KUKA KRL program: MyProgram_320().src

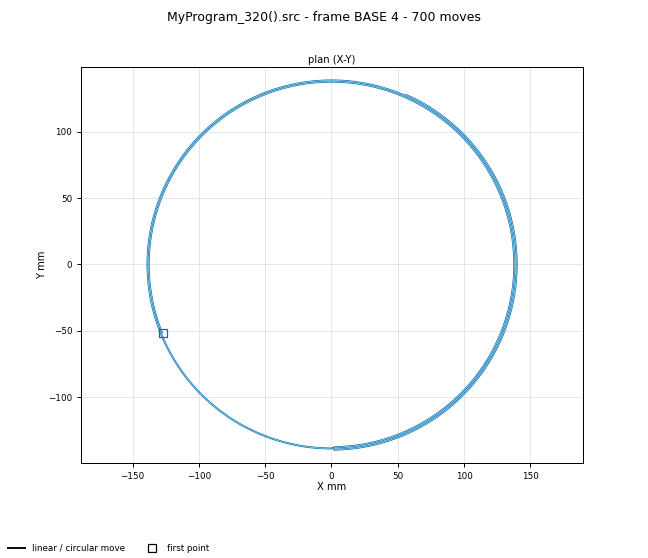
[picture p0: tool path of MyProgram_320().src in frame BASE 4, 700 of 700 moves have a stored position in this frame; points joined in program order, loops and branches not executed]
&ACCESS RVP
&REL 1
&PARAM TEMPLATE = C:\KRC\Roboter\Template\vorgabe
&PARAM EDITMASK = *
DEF MyProgram_320()
; ---- Setting reference (Base) ----
$BASE = BASE_DATA[4]

; --------------------------
; ---- Setting tool (TCP) ----
$TOOL = TOOL_DATA[3]
; --------------------------

$VEL.CP = VEL_APROX_PRINT
Startdeposition()
$VEL.CP = VEL_PRINT
LIN {X -127.2206,Y -51.8172,Z 185,A -153.9246,B 3.1278,C 0.2354,E1 2.9885,E2 247.0767} C_DIS
LIN {X -128.3074,Y -49.0677,Z 185,A -155.3949,B 3.128,C 0.2331,E1 2.987,E2 248.577} C_DIS
LIN {X -129.8881,Y -44.7108,Z 185,A -157.1036,B 3.1284,C 0.2271,E1 2.9854,E2 250.256} C_DIS
LIN {X -131.3839,Y -40.1019,Z 185,A -159.2672,B 3.1288,C 0.2223,E1 2.9836,E2 252.4369} C_DIS
LIN {X -132.2695,Y -37.0766,Z 185,A -160.5831,B 3.129,C 0.2188,E1 2.9825,E2 253.7523} C_DIS
LIN {X -133.0577,Y -34.142,Z 185,A -162.0522,B 3.1292,C 0.2162,E1 2.9815,E2 255.2465} C_DIS
LIN {X -133.9039,Y -30.6537,Z 185,A -163.578,B 3.1295,C 0.2122,E1 2.9805,E2 256.7752} C_DIS
LIN {X -134.6157,Y -27.3594,Z 185,A -164.9526,B 3.1298,C 0.2082,E1 2.9797,E2 258.145} C_DIS
LIN {X -135.1791,Y -24.4249,Z 185,A -166.2419,B 3.13,C 0.205,E1 2.979,E2 259.4392} C_DIS
LIN {X -135.7212,Y -21.207,Z 185,A -167.7582,B 3.1302,C 0.2018,E1 2.9784,E2 260.9744} C_DIS
LIN {X -136.2012,Y -17.8658,Z 185,A -169.3042,B 3.1304,C 0.1984,E1 2.9778,E2 262.5371} C_DIS
LIN {X -136.7019,Y -13.5167,Z 185,A -171.2437,B 3.1307,C 0.1937,E1 2.9772,E2 264.4899} C_DIS
LIN {X -136.999,Y -10.063,Z 185,A -172.73,B 3.1309,C 0.1898,E1 2.9768,E2 265.9804} C_DIS
LIN {X -137.2502,Y -5.6994,Z 185,A -174.6658,B 3.1312,C 0.1851,E1 2.9766,E2 267.9293} C_DIS
LIN {X -137.3622,Y -1.4594,Z 185,A -176.5532,B 3.1315,C 0.1806,E1 2.9765,E2 269.8305} C_DIS
LIN {X -137.346,Y 2.474,Z 185,A -178.1887,B 3.1317,C 0.1759,E1 2.9765,E2 271.4643} C_DIS
LIN {X -137.2122,Y 6.5512,Z 185,A 179.9992,B 3.132,C 0.1716,E1 2.9767,E2 273.2891} C_DIS
LIN {X -136.9944,Y 10.1259,Z 185,A 178.4827,B 3.1322,C 0.1674,E1 2.977,E2 274.8074} C_DIS
LIN {X -136.6818,Y 13.7268,Z 185,A 176.7446,B 3.1324,C 0.1641,E1 2.9775,E2 276.5735} C_DIS
LIN {X -136.1552,Y 18.2164,Z 185,A 174.8363,B 3.1326,C 0.1589,E1 2.9781,E2 278.4833} C_DIS
LIN {X -135.5392,Y 22.3415,Z 185,A 173.1558,B 3.1329,C 0.1538,E1 2.9789,E2 280.1551} C_DIS
LIN {X -134.953,Y 25.6446,Z 185,A 171.7399,B 3.1331,C 0.15,E1 2.9796,E2 281.5721} C_DIS
LIN {X -134.4845,Y 28.0041,Z 185,A 170.5079,B 3.1331,C 0.1481,E1 2.9803,E2 282.832} C_DIS
LIN {X -133.7699,Y 31.2406,Z 185,A 169.0156,B 3.1333,C 0.1447,E1 2.9812,E2 284.3369} C_DIS
LIN {X -132.7902,Y 35.167,Z 185,A 167.5567,B 3.1336,C 0.1392,E1 2.9822,E2 285.766} C_DIS
LIN {X -131.8831,Y 38.4286,Z 185,A 165.6724,B 3.1336,C 0.1372,E1 2.9837,E2 287.708} C_DIS
LIN {X -130.4216,Y 43.1295,Z 185,A 163.8308,B 3.1339,C 0.1309,E1 2.9852,E2 289.5218} C_DIS
LIN {X -129.6058,Y 45.525,Z 185,A 162.5514,B 3.134,C 0.1289,E1 2.9864,E2 290.8282} C_DIS
LIN {X -128.1871,Y 49.3771,Z 185,A 161.0189,B 3.1342,C 0.1238,E1 2.9879,E2 292.3371} C_DIS
LIN {X -127.3534,Y 51.4877,Z 185,A 158.726,B 3.1342,C 0.1265,E1 2.9906,E2 294.7944} C_DIS
LIN {X -124.3017,Y 58.4774,Z 185,A 156.4051,B 3.1346,C 0.1151,E1 2.9931,E2 297.0081} C_DIS
LIN {X -122.5678,Y 62.0248,Z 185,A 154.87,B 3.1347,C 0.1105,E1 2.995,E2 298.5281} C_DIS
LIN {X -120.8252,Y 65.3591,Z 185,A 153.0785,B 3.1348,C 0.1075,E1 2.9974,E2 300.3459} C_DIS
LIN {X -118.619,Y 69.2824,Z 185,A 151.1069,B 3.135,C 0.1033,E1 3.0001,E2 302.3275} C_DIS
LIN {X -116.2679,Y 73.1587,Z 185,A 149.325,B 3.1351,C 0.0984,E1 3.0027,E2 304.0945} C_DIS
LIN {X -113.2304,Y 77.7771,Z 185,A 146.7901,B 3.1353,C 0.094,E1 3.0067,E2 306.6559} C_DIS
LIN {X -110.5879,Y 81.4907,Z 185,A 144.8026,B 3.1353,C 0.0901,E1 3.0099,E2 308.6525} C_DIS
LIN {X -107.9657,Y 84.9341,Z 185,A 142.9194,B 3.1355,C 0.0865,E1 3.0132,E2 310.5437} C_DIS
LIN {X -104.5605,Y 89.0927,Z 185,A 140.5857,B 3.1355,C 0.0821,E1 3.0173,E2 312.8869} C_DIS
LIN {X -101.4653,Y 92.6032,Z 185,A 138.5535,B 3.1357,C 0.0785,E1 3.0212,E2 314.9274} C_DIS
LIN {X -98.4395,Y 95.8133,Z 185,A 136.6894,B 3.1357,C 0.0749,E1 3.0248,E2 316.793} C_DIS
LIN {X -95.2668,Y 98.9686,Z 185,A 134.7267,B 3.1358,C 0.0718,E1 3.0287,E2 318.766} C_DIS
LIN {X -92.1092,Y 101.9135,Z 185,A 132.8935,B 3.1359,C 0.0686,E1 3.0325,E2 320.6017} C_DIS
LIN {X -88.6534,Y 104.9339,Z 185,A 130.9144,B 3.1359,C 0.0655,E1 3.0367,E2 322.5872} C_DIS
LIN {X -86.0163,Y 107.1059,Z 185,A 129.2483,B 3.136,C 0.0643,E1 3.0404,E2 324.2815} C_DIS
LIN {X -83.4152,Y 109.1434,Z 185,A 128.0792,B 3.136,C 0.061,E1 3.0429,E2 325.4243} C_DIS
LIN {X -79.93,Y 111.721,Z 185,A 126.1941,B 3.1361,C 0.0585,E1 3.0472,E2 327.3174} C_DIS
LIN {X -76.2262,Y 114.2802,Z 185,A 124.3048,B 3.1361,C 0.0557,E1 3.0515,E2 329.2068} C_DIS
LIN {X -72.531,Y 116.6604,Z 185,A 122.6104,B 3.1362,C 0.0524,E1 3.0555,E2 330.8831} C_DIS
LIN {X -68.5121,Y 119.0656,Z 185,A 120.4438,B 3.1362,C 0.0509,E1 3.0608,E2 333.0742} C_DIS
LIN {X -64.7458,Y 121.1547,Z 185,A 117.9732,B 3.1362,C 0.0521,E1 3.0671,E2 335.6243} C_DIS
LIN {X -60.0472,Y 123.5509,Z 185,A 116.2413,B 3.1363,C 0.0471,E1 3.0712,E2 337.2988} C_DIS
LIN {X -56.4708,Y 125.2241,Z 185,A 114.8247,B 3.1363,C 0.0441,E1 3.0748,E2 338.6867} C_DIS
LIN {X -53.2256,Y 126.6372,Z 185,A 112.9364,B 3.1363,C 0.0449,E1 3.0798,E2 340.6235} C_DIS
LIN {X -50.1738,Y 127.8774,Z 185,A 111.996,B 3.1363,C 0.0412,E1 3.0821,E2 341.5109} C_DIS
LIN {X -47.5465,Y 128.8785,Z 185,A 110.5514,B 3.1363,C 0.0417,E1 3.0859,E2 342.9876} C_DIS
LIN {X -43.669,Y 130.242,Z 185,A 108.8857,B 3.1364,C 0.04,E1 3.0903,E2 344.6463} C_DIS
LIN {X -40.3704,Y 131.3017,Z 185,A 107.4297,B 3.1364,C 0.039,E1 3.0942,E2 346.1028} C_DIS
LIN {X -36.1258,Y 132.5345,Z 185,A 105.463,B 3.1364,C 0.0385,E1 3.0995,E2 348.0833} C_DIS
LIN {X -32.4216,Y 133.4871,Z 185,A 104.0145,B 3.1364,C 0.0367,E1 3.1034,E2 349.5132} C_DIS
LIN {X -29.6457,Y 134.1324,Z 185,A 102.663,B 3.1364,C 0.0371,E1 3.1071,E2 350.8836} C_DIS
LIN {X -25.59,Y 134.9634,Z 185,A 100.9801,B 3.1364,C 0.0361,E1 3.1117,E2 352.5604} C_DIS
LIN {X -21.1664,Y 135.7275,Z 185,A 99.211,B 3.1364,C 0.0348,E1 3.1166,E2 354.316} C_DIS
LIN {X -17.9099,Y 136.1954,Z 185,A 97.7627,B 3.1364,C 0.0349,E1 3.1206,E2 355.7728} C_DIS
LIN {X -12.6318,Y 136.7867,Z 185,A 94.5314,B 3.1364,C 0.0411,E1 3.13,E2 359.1239} C_DIS
LIN {X -5.4981,Y 137.2581,Z 185,A 92.5658,B 3.1364,C 0.0344,E1 3.1351,E2 360.9673} C_DIS
LIN {X 1.8136,Y 137.357,Z 185,A 89.5018,B 3.1364,C 0.0348,E1 3.1437,E2 364.0318} C_DIS
LIN {X 9.2316,Y 137.0596,Z 185,A 86.3024,B 3.1364,C 0.0363,E1 3.1526,E2 367.2424} C_DIS
LIN {X 15.1597,Y 136.5297,Z 185,A 83.5212,B 3.1364,C 0.0394,E1 3.1605,E2 370.0585} C_DIS
LIN {X 19.2177,Y 136.0172,Z 185,A 82.2725,B 3.1364,C 0.037,E1 3.1638,E2 371.2518} C_DIS
LIN {X 22.3777,Y 135.5331,Z 185,A 80.9467,B 3.1364,C 0.0376,E1 3.1674,E2 372.5762} C_DIS
LIN {X 25.7451,Y 134.9337,Z 185,A 79.5762,B 3.1364,C 0.0381,E1 3.1712,E2 373.9396} C_DIS
LIN {X 28.5414,Y 134.3708,Z 185,A 78.4896,B 3.1364,C 0.0381,E1 3.1741,E2 375.0134} C_DIS
LIN {X 31.7927,Y 133.6387,Z 185,A 76.9984,B 3.1364,C 0.04,E1 3.1782,E2 376.5164} C_DIS
LIN {X 35.2086,Y 132.7791,Z 185,A 75.5841,B 3.1364,C 0.0407,E1 3.182,E2 377.9236} C_DIS
LIN {X 38.3332,Y 131.9111,Z 185,A 74.2324,B 3.1364,C 0.0419,E1 3.1856,E2 379.275} C_DIS
LIN {X 41.6265,Y 130.9089,Z 185,A 72.8018,B 3.1364,C 0.0432,E1 3.1895,E2 380.7046} C_DIS
LIN {X 44.8549,Y 129.8381,Z 185,A 71.3415,B 3.1364,C 0.045,E1 3.1933,E2 382.1696} C_DIS
LIN {X 49.4529,Y 128.1577,Z 185,A 69.3854,B 3.1364,C 0.0465,E1 3.1984,E2 384.115} C_DIS
LIN {X 52.5735,Y 126.9096,Z 185,A 68.0035,B 3.1363,C 0.048,E1 3.202,E2 385.4942} C_DIS
LIN {X 55.8092,Y 125.52,Z 185,A 66.7765,B 3.1363,C 0.0479,E1 3.2051,E2 386.6917} C_DIS
LIN {X 58.9894,Y 124.0571,Z 185,A 65.1798,B 3.1363,C 0.0508,E1 3.2092,E2 388.3049} C_DIS
LIN {X 62.1187,Y 122.52,Z 185,A 63.7792,B 3.1363,C 0.0524,E1 3.2127,E2 389.6988} C_DIS
LIN {X 65.4146,Y 120.7953,Z 185,A 62.0738,B 3.1362,C 0.0558,E1 3.2169,E2 391.4229} C_DIS
LIN {X 69.3364,Y 118.5873,Z 185,A 60.2725,B 3.1362,C 0.058,E1 3.2213,E2 393.2149} C_DIS
LIN {X 73.2071,Y 116.2374,Z 185,A 58.4362,B 3.1361,C 0.0605,E1 3.2256,E2 395.0447} C_DIS
LIN {X 76.9789,Y 113.7746,Z 185,A 56.6058,B 3.1361,C 0.0632,E1 3.2299,E2 396.8692} C_DIS
LIN {X 80.6259,Y 111.2199,Z 185,A 54.8233,B 3.136,C 0.0657,E1 3.2339,E2 398.6426} C_DIS
LIN {X 84.0737,Y 108.6371,Z 185,A 53.0719,B 3.136,C 0.0685,E1 3.2378,E2 400.3886} C_DIS
LIN {X 87.511,Y 105.8878,Z 185,A 51.2684,B 3.1358,C 0.0716,E1 3.2417,E2 402.1882} C_DIS
LIN {X 91.1,Y 102.8163,Z 185,A 49.6038,B 3.1358,C 0.0727,E1 3.2451,E2 403.8156} C_DIS
LIN {X 93.7824,Y 100.3758,Z 185,A 47.9612,B 3.1358,C 0.0768,E1 3.2485,E2 405.4743} C_DIS
LIN {X 96.8021,Y 97.4666,Z 185,A 46.2566,B 3.1356,C 0.0799,E1 3.2519,E2 407.1737} C_DIS
LIN {X 99.6214,Y 94.5841,Z 185,A 44.7019,B 3.1356,C 0.0823,E1 3.2549,E2 408.7131} C_DIS
LIN {X 102.2276,Y 91.7602,Z 185,A 43.0242,B 3.1355,C 0.0864,E1 3.2581,E2 410.4003} C_DIS
LIN {X 105.1144,Y 88.4387,Z 185,A 41.2518,B 3.1354,C 0.0898,E1 3.2613,E2 412.1653} C_DIS
LIN {X 107.8952,Y 85.0239,Z 185,A 39.4783,B 3.1353,C 0.0934,E1 3.2644,E2 413.9314} C_DIS
LIN {X 110.6338,Y 81.4283,Z 185,A 37.6704,B 3.1352,C 0.097,E1 3.2674,E2 415.7303} C_DIS
LIN {X 113.1668,Y 77.8697,Z 185,A 35.9227,B 3.1351,C 0.1005,E1 3.2702,E2 417.4693} C_DIS
LIN {X 114.8292,Y 75.3968,Z 185,A 34.6044,B 3.1349,C 0.1042,E1 3.2722,E2 418.7973} C_DIS
LIN {X 116.6535,Y 72.5421,Z 185,A 32.6213,B 3.1346,C 0.113,E1 3.2753,E2 420.8509} C_DIS
LIN {X 119.8789,Y 67.0784,Z 185,A 30.7963,B 3.1346,C 0.1118,E1 3.2776,E2 422.5758} C_DIS
LIN {X 122.1471,Y 62.8512,Z 185,A 29.0018,B 3.1346,C 0.1148,E1 3.2799,E2 424.3453} C_DIS
LIN {X 123.6929,Y 59.7517,Z 185,A 27.4883,B 3.1344,C 0.1192,E1 3.2818,E2 425.8679} C_DIS
LIN {X 125.0111,Y 56.9438,Z 185,A 26.0373,B 3.1342,C 0.124,E1 3.2835,E2 427.3391} C_DIS
LIN {X 126.4267,Y 53.7295,Z 185,A 23.9921,B 3.1338,C 0.1335,E1 3.2858,E2 429.4566} C_DIS
LIN {X 129.0057,Y 47.1998,Z 185,A 22.0204,B 3.1338,C 0.1319,E1 3.2876,E2 431.311} C_DIS
LIN {X 130.2761,Y 43.5666,Z 185,A 20.5744,B 3.1338,C 0.1347,E1 3.2889,E2 432.7378} C_DIS
LIN {X 131.3256,Y 40.2925,Z 185,A 19.2721,B 3.1337,C 0.1372,E1 3.29,E2 434.0243} C_DIS
LIN {X 132.3115,Y 36.9264,Z 185,A 17.8228,B 3.1335,C 0.1411,E1 3.2911,E2 435.4725} C_DIS
LIN {X 133.1382,Y 33.8247,Z 185,A 16.5536,B 3.1334,C 0.144,E1 3.292,E2 436.7337} C_DIS
LIN {X 133.8617,Y 30.8387,Z 185,A 15.3424,B 3.1332,C 0.1469,E1 3.2928,E2 437.9367} C_DIS
LIN {X 134.4778,Y 28.0373,Z 185,A 14.0616,B 3.133,C 0.151,E1 3.2935,E2 439.2289} C_DIS
LIN {X 135.2029,Y 24.2921,Z 185,A 12.5685,B 3.1329,C 0.1544,E1 3.2943,E2 440.7104} C_DIS
LIN {X 135.9145,Y 19.9358,Z 185,A 11.0001,B 3.1327,C 0.1568,E1 3.2949,E2 442.2454} C_DIS
LIN {X 136.6326,Y 14.2037,Z 185,A 8.465,B 3.1323,C 0.1649,E1 3.2958,E2 444.7979} C_DIS
LIN {X 137.239,Y 5.9882,Z 185,A 5.1999,B 3.1319,C 0.1728,E1 3.2964,E2 448.0435} C_DIS
LIN {X 137.352,Y 2.1098,Z 185,A 3.8317,B 3.1318,C 0.1748,E1 3.2964,E2 449.3808} C_DIS
LIN {X 137.3445,Y -2.5652,Z 185,A 1.3682,B 3.1312,C 0.1855,E1 3.2964,E2 451.9109} C_DIS
LIN {X 137.1832,Y -7.1289,Z 185,A -0.0422,B 3.1312,C 0.1859,E1 3.2962,E2 453.2598} C_DIS
LIN {X 136.8906,Y -11.443,Z 185,A -1.7494,B 3.1309,C 0.19,E1 3.2958,E2 454.9559} C_DIS
LIN {X 136.4657,Y -15.7279,Z 185,A -3.9041,B 3.1304,C 0.1987,E1 3.2952,E2 457.1577} C_DIS
LIN {X 135.8556,Y -20.3391,Z 185,A -5.3709,B 3.1304,C 0.1993,E1 3.2946,E2 458.5656} C_DIS
LIN {X 135.2516,Y -24.02,Z 185,A -6.7383,B 3.1302,C 0.2018,E1 3.294,E2 459.9098} C_DIS
LIN {X 134.7097,Y -26.8975,Z 185,A -7.7917,B 3.1301,C 0.2035,E1 3.2934,E2 460.9425} C_DIS
LIN {X 133.992,Y -30.2682,Z 185,A -9.2727,B 3.1298,C 0.2079,E1 3.2925,E2 462.4302} C_DIS
LIN {X 133.1727,Y -33.6888,Z 185,A -10.7278,B 3.1295,C 0.2118,E1 3.2916,E2 463.8848} C_DIS
LIN {X 132.2958,Y -36.9825,Z 185,A -11.9845,B 3.1294,C 0.214,E1 3.2907,E2 465.1212} C_DIS
LIN {X 131.4704,Y -39.8192,Z 185,A -13.3051,B 3.1291,C 0.2183,E1 3.2896,E2 466.4543} C_DIS
LIN {X 130.5719,Y -42.6782,Z 185,A -14.4871,B 3.1289,C 0.221,E1 3.2886,E2 467.6285} C_DIS
LIN {X 129.3343,Y -46.2882,Z 185,A -15.9446,B 3.1287,C 0.2239,E1 3.2873,E2 469.0698} C_DIS
LIN {X 128.1113,Y -49.5722,Z 185,A -17.3701,B 3.1284,C 0.2274,E1 3.2859,E2 470.4918} C_DIS
LIN {X 126.7284,Y -53.0073,Z 185,A -18.8286,B 3.1282,C 0.2306,E1 3.2843,E2 471.9402} C_DIS
LIN {X 125.6739,Y -55.465,Z 185,A -19.9685,B 3.1279,C 0.2338,E1 3.283,E2 473.0843} C_DIS
LIN {X 124.0202,Y -59.0665,Z 185,A -21.4912,B 3.1277,C 0.2368,E1 3.2813,E2 474.5913} C_DIS
LIN {X 122.6016,Y -61.9584,Z 185,A -22.7609,B 3.1275,C 0.2395,E1 3.2797,E2 475.8526} C_DIS
LIN {X 120.8252,Y -65.3591,Z 185,A -24.7938,B 3.1269,C 0.2478,E1 3.2769,E2 477.943} C_DIS
LIN {X 118.6705,Y -69.1946,Z 185,A -26.2059,B 3.1269,C 0.2482,E1 3.275,E2 479.3017} C_DIS
LIN {X 116.4356,Y -72.8922,Z 185,A -27.8995,B 3.1266,C 0.2515,E1 3.2726,E2 480.9826} C_DIS
LIN {X 114.5094,Y -75.8825,Z 185,A -29.7412,B 3.126,C 0.2586,E1 3.2697,E2 482.8721} C_DIS
LIN {X 111.9579,Y -79.5988,Z 185,A -31.1758,B 3.126,C 0.2587,E1 3.2674,E2 484.2502} C_DIS
LIN {X 109.3387,Y -83.16,Z 185,A -32.9566,B 3.1257,C 0.2624,E1 3.2645,E2 486.0242} C_DIS
LIN {X 106.5413,Y -86.7146,Z 185,A -34.8528,B 3.1253,C 0.2668,E1 3.2612,E2 487.9233} C_DIS
LIN {X 103.8669,Y -89.9008,Z 185,A -36.8226,B 3.1248,C 0.2728,E1 3.2575,E2 489.9251} C_DIS
LIN {X 100.8615,Y -93.2604,Z 185,A -38.2429,B 3.1248,C 0.2725,E1 3.2549,E2 491.2868} C_DIS
LIN {X 97.7188,Y -96.5482,Z 185,A -40.1537,B 3.1245,C 0.2766,E1 3.2512,E2 493.201} C_DIS
LIN {X 94.2509,Y -99.9358,Z 185,A -42.0108,B 3.1242,C 0.2792,E1 3.2475,E2 495.038} C_DIS
LIN {X 90.5016,Y -103.3437,Z 185,A -44.0948,B 3.1239,C 0.2831,E1 3.2432,E2 497.1198} C_DIS
LIN {X 87.0714,Y -106.2497,Z 185,A -45.9866,B 3.1235,C 0.2868,E1 3.2391,E2 499.0153} C_DIS
LIN {X 83.0844,Y -109.3963,Z 185,A -47.8812,B 3.1234,C 0.2886,E1 3.235,E2 500.8821} C_DIS
LIN {X 79.2752,Y -112.1867,Z 185,A -49.8775,B 3.123,C 0.2924,E1 3.2304,E2 502.8834} C_DIS
LIN {X 75.5788,Y -114.7094,Z 185,A -51.6453,B 3.1228,C 0.2946,E1 3.2264,E2 504.6396} C_DIS
LIN {X 72.2271,Y -116.8495,Z 185,A -53.152,B 3.1227,C 0.2959,E1 3.2228,E2 506.1275} C_DIS
LIN {X 66.1107,Y -120.4156,Z 185,A -56.0363,B 3.1223,C 0.2999,E1 3.2159,E2 509.005} C_DIS
LIN {X 62.9846,Y -122.0792,Z 185,A -57.6575,B 3.122,C 0.3032,E1 3.2118,E2 510.6463} C_DIS
LIN {X 59.3361,Y -123.8914,Z 185,A -59.2521,B 3.1218,C 0.3046,E1 3.2078,E2 512.2282} C_DIS
LIN {X 55.6679,Y -125.5832,Z 185,A -60.9267,B 3.1216,C 0.3067,E1 3.2036,E2 513.9027} C_DIS
LIN {X 51.6723,Y -127.279,Z 185,A -62.5593,B 3.1216,C 0.3074,E1 3.1994,E2 515.5129} C_DIS
LIN {X 48.9659,Y -128.3467,Z 185,A -63.9601,B 3.1213,C 0.3104,E1 3.1957,E2 516.9395} C_DIS
LIN {X 45.2189,Y -129.7119,Z 185,A -65.5888,B 3.1211,C 0.312,E1 3.1914,E2 518.5646} C_DIS
LIN {X 40.8738,Y -131.1477,Z 185,A -67.3488,B 3.1211,C 0.3126,E1 3.1868,E2 520.3062} C_DIS
LIN {X 36.9918,Y -132.2932,Z 185,A -68.9133,B 3.1211,C 0.3132,E1 3.1826,E2 521.8553} C_DIS
LIN {X 33.931,Y -133.1113,Z 185,A -70.292,B 3.1208,C 0.3148,E1 3.1789,E2 523.2424} C_DIS
LIN {X 30.5431,Y -133.9292,Z 185,A -71.7431,B 3.1208,C 0.316,E1 3.1749,E2 524.6941} C_DIS
LIN {X 26.6507,Y -134.7599,Z 185,A -73.4339,B 3.1206,C 0.3174,E1 3.1703,E2 526.39} C_DIS
LIN {X 23.6785,Y -135.3127,Z 185,A -75.6824,B 3.1197,C 0.326,E1 3.1638,E2 528.7694} C_DIS
LIN {X 16.2323,Y -136.4055,Z 185,A -77.6627,B 3.1205,C 0.3187,E1 3.1587,E2 530.5987} C_DIS
LIN {X 9.1529,Y -137.0646,Z 185,A -80.9036,B 3.1201,C 0.322,E1 3.1495,E2 533.8778} C_DIS
LIN {X 2.2312,Y -137.35,Z 185,A -83.5784,B 3.1201,C 0.3211,E1 3.1421,E2 536.5256} C_DIS
LIN {X 2.2312,Y -137.35,Z 185,A -83.5784,B 3.1201,C 0.3211,E1 3.1421,E2 536.5256} C_DIS
Enddeposition()
LIN {X 0.9813,Y -138.2634,Z 185,A -83.5483,B 3.1297,C 0.3191,E1 3.1516,E2 536.4499} C_DIS
Startdeposition()
$VEL.CP = VEL_PRINT
LIN {X 4.1352,Y -138.2067,Z 185,A -82.1164,B 3.1298,C 0.3178,E1 3.1557,E2 535.0005} C_DIS
LIN {X 7.7208,Y -138.0547,Z 185,A -80.675,B 3.1298,C 0.3178,E1 3.1597,E2 533.5646} C_DIS
LIN {X 10.8511,Y -137.844,Z 185,A -79.3806,B 3.1299,C 0.3173,E1 3.1633,E2 532.2704} C_DIS
LIN {X 14.4758,Y -137.5087,Z 185,A -77.875,B 3.1299,C 0.3167,E1 3.1675,E2 530.7643} C_DIS
LIN {X 17.1717,Y -137.2,Z 185,A -76.7623,B 3.13,C 0.3162,E1 3.1706,E2 529.6526} C_DIS
LIN {X 20.8522,Y -136.687,Z 185,A -75.2123,B 3.1301,C 0.3152,E1 3.1748,E2 528.1002} C_DIS
LIN {X 25.6575,Y -135.867,Z 185,A -73.2312,B 3.1302,C 0.3142,E1 3.1803,E2 526.1233} C_DIS
LIN {X 28.873,Y -135.2201,Z 185,A -71.8856,B 3.1303,C 0.3133,E1 3.184,E2 524.7786} C_DIS
LIN {X 32.1482,Y -134.4789,Z 185,A -70.5233,B 3.1303,C 0.3125,E1 3.1877,E2 523.4194} C_DIS
LIN {X 35.3199,Y -133.681,Z 185,A -69.171,B 3.1305,C 0.3113,E1 3.1913,E2 522.0667} C_DIS
LIN {X 38.0462,Y -132.933,Z 185,A -67.8723,B 3.1307,C 0.3092,E1 3.1949,E2 520.7501} C_DIS
LIN {X 41.7685,Y -131.8085,Z 185,A -66.5596,B 3.1307,C 0.3101,E1 3.1983,E2 519.4767} C_DIS
LIN {X 44.4883,Y -130.9179,Z 185,A -65.2589,B 3.1308,C 0.3079,E1 3.2018,E2 518.1597} C_DIS
LIN {X 48.0865,Y -129.6374,Z 185,A -63.6729,B 3.131,C 0.3061,E1 3.2059,E2 516.5721} C_DIS
LIN {X 51.3902,Y -128.3633,Z 185,A -62.2604,B 3.1311,C 0.3049,E1 3.2096,E2 515.1661} C_DIS
LIN {X 54.6278,Y -127.0191,Z 185,A -60.8496,B 3.1313,C 0.3035,E1 3.2132,E2 513.7599} C_DIS
LIN {X 57.7327,Y -125.6384,Z 185,A -59.6462,B 3.1313,C 0.3035,E1 3.2162,E2 512.583} C_DIS
LIN {X 60.3884,Y -124.3863,Z 185,A -58.2622,B 3.1316,C 0.3003,E1 3.2198,E2 511.1758} C_DIS
LIN {X 63.5069,Y -122.8234,Z 185,A -56.7072,B 3.1319,C 0.2973,E1 3.2237,E2 509.6048} C_DIS
LIN {X 67.3646,Y -120.7507,Z 185,A -54.953,B 3.1321,C 0.2952,E1 3.228,E2 507.8575} C_DIS
LIN {X 71.1713,Y -118.5469,Z 185,A -53.1835,B 3.1323,C 0.2928,E1 3.2322,E2 506.0939} C_DIS
LIN {X 74.9206,Y -116.2137,Z 185,A -51.5093,B 3.1324,C 0.2912,E1 3.2361,E2 504.4393} C_DIS
LIN {X 78.1008,Y -114.1,Z 185,A -49.9155,B 3.1327,C 0.2885,E1 3.2398,E2 502.8427} C_DIS
LIN {X 81.5037,Y -111.6954,Z 185,A -48.2879,B 3.1329,C 0.2864,E1 3.2435,E2 501.2271} C_DIS
LIN {X 84.5715,Y -109.3902,Z 185,A -46.6821,B 3.1332,C 0.2833,E1 3.247,E2 499.618} C_DIS
LIN {X 87.8428,Y -106.7818,Z 185,A -45.0586,B 3.1334,C 0.2811,E1 3.2505,E2 498.0079} C_DIS
LIN {X 90.9521,Y -104.1452,Z 185,A -43.3668,B 3.1336,C 0.2778,E1 3.2541,E2 496.3144} C_DIS
LIN {X 94.1057,Y -101.3048,Z 185,A -41.7154,B 3.1339,C 0.2753,E1 3.2575,E2 494.676} C_DIS
LIN {X 96.9393,Y -98.5967,Z 185,A -40.1086,B 3.1341,C 0.2722,E1 3.2607,E2 493.0703} C_DIS
LIN {X 99.6517,Y -95.8553,Z 185,A -38.5217,B 3.1344,C 0.2689,E1 3.2638,E2 491.4836} C_DIS
LIN {X 102.6999,Y -92.5821,Z 185,A -36.7443,B 3.1347,C 0.2657,E1 3.2672,E2 489.7149} C_DIS
LIN {X 105.5902,Y -89.2713,Z 185,A -34.9767,B 3.135,C 0.2622,E1 3.2704,E2 487.953} C_DIS
LIN {X 108.0789,Y -86.2409,Z 185,A -33.3908,B 3.1353,C 0.2589,E1 3.2731,E2 486.371} C_DIS
LIN {X 110.8016,Y -82.7136,Z 185,A -31.7,B 3.1355,C 0.2562,E1 3.276,E2 484.6994} C_DIS
LIN {X 113.1584,Y -79.4592,Z 185,A -30.0798,B 3.1358,C 0.2527,E1 3.2786,E2 483.0839} C_DIS
LIN {X 115.5333,Y -75.9643,Z 185,A -28.3636,B 3.1361,C 0.2488,E1 3.2813,E2 481.3709} C_DIS
LIN {X 117.9476,Y -72.1589,Z 185,A -26.5817,B 3.1364,C 0.2451,E1 3.2839,E2 479.5988} C_DIS
LIN {X 120.0197,Y -68.6573,Z 185,A -24.9011,B 3.1367,C 0.241,E1 3.2862,E2 477.9177} C_DIS
LIN {X 122.0101,Y -65.0556,Z 185,A -23.3573,B 3.1369,C 0.2383,E1 3.2883,E2 476.3939} C_DIS
LIN {X 123.6155,Y -61.951,Z 185,A -21.9277,B 3.1372,C 0.2348,E1 3.2901,E2 474.9657} C_DIS
LIN {X 125.1925,Y -58.697,Z 185,A -20.5769,B 3.1373,C 0.2324,E1 3.2917,E2 473.6332} C_DIS
LIN {X 126.5706,Y -55.665,Z 185,A -19.2064,B 3.1376,C 0.2289,E1 3.2932,E2 472.2629} C_DIS
LIN {X 128.0273,Y -52.2237,Z 185,A -17.6568,B 3.1379,C 0.2248,E1 3.2949,E2 470.7118} C_DIS
LIN {X 129.3689,Y -48.8034,Z 185,A -16.2643,B 3.1381,C 0.2221,E1 3.2963,E2 469.3353} C_DIS
LIN {X 130.5335,Y -45.5971,Z 185,A -14.9108,B 3.1383,C 0.2189,E1 3.2975,E2 467.9887} C_DIS
LIN {X 131.4535,Y -42.88,Z 185,A -13.7724,B 3.1385,C 0.2163,E1 3.2985,E2 466.856} C_DIS
LIN {X 132.6072,Y -39.1592,Z 185,A -12.3657,B 3.1386,C 0.214,E1 3.2997,E2 465.4753} C_DIS
LIN {X 133.5161,Y -35.9382,Z 185,A -11.0797,B 3.1388,C 0.2112,E1 3.3006,E2 464.2015} C_DIS
LIN {X 134.2236,Y -33.2077,Z 185,A -9.7375,B 3.1392,C 0.2063,E1 3.3015,E2 462.8359} C_DIS
LIN {X 134.9802,Y -29.9843,Z 185,A -8.4715,B 3.1393,C 0.2035,E1 3.3023,E2 461.5827} C_DIS
LIN {X 135.655,Y -26.7663,Z 185,A -7.0347,B 3.1396,C 0.199,E1 3.3031,E2 460.1352} C_DIS
LIN {X 136.3318,Y -23.0605,Z 185,A -5.8526,B 3.1396,C 0.1985,E1 3.3037,E2 459.0014} C_DIS
LIN {X 136.8342,Y -19.8635,Z 185,A -4.3967,B 3.14,C 0.1936,E1 3.3043,E2 457.5295} C_DIS
LIN {X 137.2,Y -17.1717,Z 185,A -3.1895,B 3.1402,C 0.1896,E1 3.3047,E2 456.311} C_DIS
LIN {X 137.6065,Y -13.5135,Z 185,A -1.8645,B 3.1403,C 0.1874,E1 3.3051,E2 455.011} C_DIS
LIN {X 137.8941,Y -10.1646,Z 185,A -0.5282,B 3.1405,C 0.1841,E1 3.3054,E2 453.6812} C_DIS
LIN {X 138.133,Y -6.1641,Z 185,A 1.1793,B 3.1408,C 0.1789,E1 3.3056,E2 451.9664} C_DIS
LIN {X 138.2364,Y -3.069,Z 185,A 2.2773,B 3.1409,C 0.1772,E1 3.3057,E2 450.8918} C_DIS
LIN {X 138.2715,Y 0,Z 185,A 3.6446,B 3.1412,C 0.1726,E1 3.3057,E2 449.5112} C_DIS
LIN {X 138.2206,Y 3.6378,Z 185,A 4.9795,B 3.1413,C 0.1701,E1 3.3057,E2 448.1977} C_DIS
LIN {X 138.0547,Y 7.7208,Z 185,A 6.561,B 3.1415,C 0.1665,E1 3.3054,E2 446.6297} C_DIS
LIN {X 137.844,Y 10.8511,Z 185,A 7.9221,B 3.1417,C 0.1622,E1 3.3052,E2 445.2599} C_DIS
LIN {X 137.5596,Y 14.0022,Z 185,A 9.1962,B 3.1419,C 0.1589,E1 3.3048,E2 443.9898} C_DIS
LIN {X 137.2,Y 17.1717,Z 185,A 10.331,B 3.142,C 0.1571,E1 3.3044,E2 442.8784} C_DIS
LIN {X 136.687,Y 20.8522,Z 185,A 11.6316,B 3.142,C 0.1553,E1 3.3039,E2 441.6077} C_DIS
LIN {X 136.2491,Y 23.5563,Z 185,A 13.0309,B 3.1424,C 0.1494,E1 3.3033,E2 440.1738} C_DIS
LIN {X 135.5537,Y 27.2643,Z 185,A 14.3949,B 3.1424,C 0.1471,E1 3.3026,E2 438.8346} C_DIS
LIN {X 134.8662,Y 30.4833,Z 185,A 15.7031,B 3.1426,C 0.1439,E1 3.3018,E2 437.5327} C_DIS
LIN {X 134.0839,Y 33.7581,Z 185,A 17.0594,B 3.1428,C 0.1405,E1 3.3009,E2 436.1807} C_DIS
LIN {X 133.2444,Y 36.9329,Z 185,A 18.1644,B 3.1428,C 0.1393,E1 3.3001,E2 435.1078} C_DIS
LIN {X 132.3083,Y 40.1576,Z 185,A 19.7036,B 3.1431,C 0.1341,E1 3.2989,E2 433.549} C_DIS
LIN {X 131.3838,Y 43.0893,Z 185,A 20.9229,B 3.1431,C 0.1312,E1 3.2978,E2 432.3361} C_DIS
LIN {X 130.361,Y 46.0946,Z 185,A 22.1669,B 3.1433,C 0.1284,E1 3.2967,E2 431.1007} C_DIS
LIN {X 129.1832,Y 49.2991,Z 185,A 23.5257,B 3.1434,C 0.1252,E1 3.2954,E2 429.7484} C_DIS
LIN {X 127.72,Y 52.9687,Z 185,A 25.1028,B 3.1436,C 0.1215,E1 3.2937,E2 428.1782} C_DIS
LIN {X 126.3518,Y 56.1543,Z 185,A 26.4787,B 3.1437,C 0.1184,E1 3.2922,E2 426.8094} C_DIS
LIN {X 125.1358,Y 58.8196,Z 185,A 27.6454,B 3.1438,C 0.1157,E1 3.2908,E2 425.6483} C_DIS
LIN {X 123.6155,Y 61.951,Z 185,A 29.164,B 3.144,C 0.1113,E1 3.2889,E2 424.1194} C_DIS
LIN {X 121.5956,Y 65.8272,Z 185,A 30.8934,B 3.144,C 0.1076,E1 3.2867,E2 422.3998} C_DIS
LIN {X 119.444,Y 69.6551,Z 185,A 32.5882,B 3.1442,C 0.1043,E1 3.2843,E2 420.7202} C_DIS
LIN {X 117.1623,Y 73.4282,Z 185,A 34.3479,B 3.1443,C 0.1005,E1 3.2818,E2 418.9685} C_DIS
LIN {X 114.905,Y 76.9115,Z 185,A 35.9765,B 3.1444,C 0.0973,E1 3.2793,E2 417.3509} C_DIS
LIN {X 112.7343,Y 80.0606,Z 185,A 37.5703,B 3.1445,C 0.0935,E1 3.2767,E2 415.7556} C_DIS
LIN {X 110.1005,Y 83.6456,Z 185,A 39.2489,B 3.1446,C 0.0908,E1 3.2739,E2 414.0973} C_DIS
LIN {X 107.9069,Y 86.457,Z 185,A 40.6753,B 3.1446,C 0.088,E1 3.2715,E2 412.6771} C_DIS
LIN {X 105.6382,Y 89.2148,Z 185,A 42.2022,B 3.1448,C 0.0843,E1 3.2687,E2 411.1439} C_DIS
LIN {X 102.6999,Y 92.5821,Z 185,A 43.9583,B 3.1448,C 0.0812,E1 3.2655,E2 409.3995} C_DIS
LIN {X 100.0785,Y 95.4088,Z 185,A 45.5225,B 3.145,C 0.0781,E1 3.2625,E2 407.8391} C_DIS
LIN {X 96.9095,Y 98.6259,Z 185,A 47.3032,B 3.145,C 0.0751,E1 3.259,E2 406.0696} C_DIS
LIN {X 93.903,Y 101.4936,Z 185,A 48.9832,B 3.1451,C 0.0721,E1 3.2556,E2 404.3946} C_DIS
LIN {X 90.7812,Y 104.2944,Z 185,A 50.6644,B 3.1451,C 0.0692,E1 3.2521,E2 402.7202} C_DIS
LIN {X 87.6287,Y 106.9568,Z 185,A 52.2637,B 3.1452,C 0.067,E1 3.2487,E2 401.1347} C_DIS
LIN {X 84.437,Y 109.4944,Z 185,A 53.9882,B 3.1452,C 0.0637,E1 3.2449,E2 399.4057} C_DIS
LIN {X 80.7836,Y 112.2173,Z 185,A 55.7406,B 3.1453,C 0.0616,E1 3.241,E2 397.6703} C_DIS
LIN {X 77.8742,Y 114.2555,Z 185,A 57.2369,B 3.1453,C 0.0589,E1 3.2375,E2 396.1709} C_DIS
LIN {X 74.1904,Y 116.6811,Z 185,A 58.955,B 3.1454,C 0.0569,E1 3.2335,E2 394.4665} C_DIS
LIN {X 70.9369,Y 118.6866,Z 185,A 60.5937,B 3.1454,C 0.054,E1 3.2296,E2 392.8209} C_DIS
LIN {X 66.8346,Y 121.0441,Z 185,A 62.4836,B 3.1455,C 0.0517,E1 3.225,E2 390.9399} C_DIS
LIN {X 63.182,Y 122.9888,Z 185,A 63.9554,B 3.1455,C 0.0513,E1 3.2214,E2 389.4984} C_DIS
LIN {X 60.3884,Y 124.3863,Z 185,A 65.3522,B 3.1455,C 0.0487,E1 3.2179,E2 388.0891} C_DIS
LIN {X 57.245,Y 125.8639,Z 185,A 66.8749,B 3.1455,C 0.0462,E1 3.214,E2 386.5562} C_DIS
LIN {X 54.08,Y 127.2559,Z 185,A 68.1647,B 3.1455,C 0.0457,E1 3.2107,E2 385.2843} C_DIS
LIN {X 50.8966,Y 128.5622,Z 185,A 69.6994,B 3.1456,C 0.0431,E1 3.2067,E2 383.7364} C_DIS
LIN {X 47.2017,Y 129.9619,Z 185,A 71.1698,B 3.1456,C 0.0427,E1 3.2029,E2 382.2868} C_DIS
LIN {X 43.9902,Y 131.0838,Z 185,A 72.3654,B 3.1456,C 0.043,E1 3.1998,E2 381.1179} C_DIS
LIN {X 41.2699,Y 131.9678,Z 185,A 73.8648,B 3.1456,C 0.0394,E1 3.1957,E2 379.5801} C_DIS
LIN {X 37.4319,Y 133.1049,Z 185,A 75.3084,B 3.1456,C 0.0395,E1 3.1919,E2 378.1633} C_DIS
LIN {X 34.4019,Y 133.9204,Z 185,A 76.5045,B 3.1456,C 0.0393,E1 3.1887,E2 376.9804} C_DIS
LIN {X 31.5955,Y 134.6122,Z 185,A 77.8163,B 3.1457,C 0.0375,E1 3.1851,E2 375.6549} C_DIS
LIN {X 28.3744,Y 135.3278,Z 185,A 79.1662,B 3.1457,C 0.0366,E1 3.1815,E2 374.3075} C_DIS
LIN {X 24.6634,Y 136.0509,Z 185,A 80.7492,B 3.1457,C 0.0355,E1 3.1771,E2 372.723} C_DIS
LIN {X 21.6068,Y 136.5702,Z 185,A 82.0235,B 3.1457,C 0.0349,E1 3.1736,E2 371.4504} C_DIS
LIN {X 18.27,Y 137.0561,Z 185,A 83.1873,B 3.1457,C 0.0359,E1 3.1704,E2 370.3156} C_DIS
LIN {X 15.0947,Y 137.4421,Z 185,A 84.6818,B 3.1457,C 0.0341,E1 3.1662,E2 368.8009} C_DIS
LIN {X 11.937,Y 137.7523,Z 185,A 86.0391,B 3.1457,C 0.0333,E1 3.1624,E2 367.4388} C_DIS
LIN {X 8.7129,Y 137.9936,Z 185,A 87.2953,B 3.1457,C 0.0334,E1 3.159,E2 366.1934} C_DIS
LIN {X 4.1352,Y 138.2067,Z 185,A 89.03,B 3.1457,C 0.0341,E1 3.1542,E2 364.4797} C_DIS
LIN {X 1.5311,Y 138.262,Z 185,A 90.4136,B 3.1457,C 0.0319,E1 3.1502,E2 363.0592} C_DIS
LIN {X -2.0074,Y 138.254,Z 185,A 91.7977,B 3.1457,C 0.0323,E1 3.1464,E2 361.6858} C_DIS
LIN {X -6.1641,Y 138.133,Z 185,A 93.4721,B 3.1457,C 0.0326,E1 3.1417,E2 360.0182} C_DIS
LIN {X -9.2832,Y 137.9584,Z 185,A 94.7702,B 3.1457,C 0.0326,E1 3.1381,E2 358.7203} C_DIS
LIN {X -12.4242,Y 137.7111,Z 185,A 96.0806,B 3.1457,C 0.0328,E1 3.1344,E2 357.4099} C_DIS
LIN {X -16.0763,Y 137.3307,Z 185,A 97.426,B 3.1457,C 0.0342,E1 3.1308,E2 356.0868} C_DIS
LIN {X -19.3229,Y 136.9114,Z 185,A 98.9581,B 3.1457,C 0.0334,E1 3.1265,E2 354.5339} C_DIS
LIN {X -21.9553,Y 136.5162,Z 185,A 100.0852,B 3.1457,C 0.0336,E1 3.1233,E2 353.4044} C_DIS
LIN {X -25.6575,Y 135.867,Z 185,A 101.6555,B 3.1457,C 0.0341,E1 3.119,E2 351.8334} C_DIS
LIN {X -28.873,Y 135.2201,Z 185,A 103.0272,B 3.1457,C 0.0347,E1 3.1153,E2 350.4608} C_DIS
LIN {X -32.0948,Y 134.4918,Z 185,A 104.4096,B 3.1457,C 0.0353,E1 3.1115,E2 349.0775} C_DIS
LIN {X -35.3199,Y 133.681,Z 185,A 105.8033,B 3.1457,C 0.036,E1 3.1077,E2 347.6827} C_DIS
LIN {X -38.0462,Y 132.933,Z 185,A 107.1375,B 3.1457,C 0.0358,E1 3.1041,E2 346.3293} C_DIS
LIN {X -41.7685,Y 131.8085,Z 185,A 108.5814,B 3.1457,C 0.038,E1 3.1003,E2 344.9068} C_DIS
LIN {X -45.0192,Y 130.7339,Z 185,A 109.85,B 3.1457,C 0.04,E1 3.097,E2 343.6575} C_DIS
LIN {X -47.6983,Y 129.7828,Z 185,A 111.2566,B 3.1457,C 0.0397,E1 3.0932,E2 342.2236} C_DIS
LIN {X -50.8966,Y 128.5622,Z 185,A 112.6982,B 3.1457,C 0.0408,E1 3.0894,E2 340.7801} C_DIS
LIN {X -54.08,Y 127.2559,Z 185,A 114.1491,B 3.1457,C 0.0421,E1 3.0857,E2 339.3271} C_DIS
LIN {X -57.3476,Y 125.8164,Z 185,A 115.6283,B 3.1457,C 0.0437,E1 3.0819,E2 337.8488} C_DIS
LIN {X -60.3884,Y 124.3863,Z 185,A 117.0757,B 3.1457,C 0.0449,E1 3.0782,E2 336.3956} C_DIS
LIN {X -63.5643,Y 122.7932,Z 185,A 118.6847,B 3.1456,C 0.0459,E1 3.0742,E2 334.7707} C_DIS
LIN {X -67.4428,Y 120.7067,Z 185,A 120.5488,B 3.1456,C 0.048,E1 3.0696,E2 332.903} C_DIS
LIN {X -71.1713,Y 118.5469,Z 185,A 122.337,B 3.1456,C 0.0504,E1 3.0653,E2 331.1157} C_DIS
LIN {X -74.6899,Y 116.3614,Z 185,A 124.0645,B 3.1455,C 0.0528,E1 3.0612,E2 329.3881} C_DIS
LIN {X -78.1008,Y 114.1,Z 185,A 125.841,B 3.1455,C 0.0549,E1 3.0571,E2 327.6028} C_DIS
LIN {X -81.5037,Y 111.6954,Z 185,A 127.5397,B 3.1454,C 0.0578,E1 3.0533,E2 325.9088} C_DIS
LIN {X -84.5715,Y 109.3902,Z 185,A 129.2384,B 3.1454,C 0.0598,E1 3.0495,E2 324.1977} C_DIS
LIN {X -87.8428,Y 106.7818,Z 185,A 130.9576,B 3.1454,C 0.0629,E1 3.0457,E2 322.4817} C_DIS
LIN {X -90.9756,Y 104.1247,Z 185,A 132.7622,B 3.1452,C 0.0654,E1 3.0419,E2 320.6657} C_DIS
LIN {X -94.1057,Y 101.3048,Z 185,A 134.5107,B 3.1452,C 0.0686,E1 3.0383,E2 318.9181} C_DIS
LIN {X -96.9864,Y 98.5505,Z 185,A 136.2417,B 3.1452,C 0.0714,E1 3.0348,E2 317.1785} C_DIS
LIN {X -99.6517,Y 95.8553,Z 185,A 137.9304,B 3.1451,C 0.0739,E1 3.0315,E2 315.4764} C_DIS
LIN {X -102.6999,Y 92.5821,Z 185,A 139.754,B 3.145,C 0.0778,E1 3.028,E2 313.6579} C_DIS
LIN {X -105.2388,Y 89.6847,Z 185,A 141.4061,B 3.1449,C 0.0809,E1 3.025,E2 312} C_DIS
LIN {X -107.5202,Y 86.9365,Z 185,A 142.9391,B 3.1449,C 0.0838,E1 3.0223,E2 310.4616} C_DIS
LIN {X -110.0516,Y 83.7095,Z 185,A 144.8051,B 3.1447,C 0.0868,E1 3.0191,E2 308.5761} C_DIS
LIN {X -112.7343,Y 80.0606,Z 185,A 146.648,B 3.1447,C 0.0912,E1 3.0161,E2 306.739} C_DIS
LIN {X -114.905,Y 76.9115,Z 185,A 148.3581,B 3.1445,C 0.0943,E1 3.0134,E2 305.0143} C_DIS
LIN {X -117.1623,Y 73.4282,Z 185,A 150.2113,B 3.1445,C 0.0977,E1 3.0106,E2 303.1458} C_DIS
LIN {X -119.444,Y 69.6551,Z 185,A 152.0487,B 3.1443,C 0.1021,E1 3.0079,E2 301.3086} C_DIS
LIN {X -121.5956,Y 65.8272,Z 185,A 153.9987,B 3.1441,C 0.106,E1 3.0053,E2 299.3435} C_DIS
LIN {X -123.4355,Y 62.3045,Z 185,A 155.6171,B 3.1441,C 0.1102,E1 3.0032,E2 297.7299} C_DIS
LIN {X -125.1358,Y 58.8196,Z 185,A 157.2632,B 3.1439,C 0.1141,E1 3.0012,E2 296.0802} C_DIS
LIN {X -126.5706,Y 55.665,Z 185,A 158.7601,B 3.1437,C 0.1175,E1 2.9995,E2 294.5767} C_DIS
LIN {X -127.9198,Y 52.4904,Z 185,A 160.2509,B 3.1437,C 0.121,E1 2.9979,E2 293.0793} C_DIS
LIN {X -129.3495,Y 48.8552,Z 185,A 161.9539,B 3.1435,C 0.1249,E1 2.9962,E2 291.3668} C_DIS
LIN {X -130.5335,Y 45.5971,Z 185,A 163.4381,B 3.1433,C 0.1285,E1 2.9948,E2 289.8776} C_DIS
LIN {X -131.4535,Y 42.88,Z 185,A 164.7753,B 3.1432,C 0.1311,E1 2.9936,E2 288.5226} C_DIS
LIN {X -132.6072,Y 39.1592,Z 185,A 166.1651,B 3.143,C 0.1363,E1 2.9925,E2 287.1624} C_DIS
LIN {X -133.5166,Y 35.9365,Z 185,A 167.8152,B 3.1429,C 0.139,E1 2.9913,E2 285.4801} C_DIS
LIN {X -134.3477,Y 32.6926,Z 185,A 169.0608,B 3.1427,C 0.1434,E1 2.9904,E2 284.2535} C_DIS
LIN {X -134.9802,Y 29.9843,Z 185,A 170.4699,B 3.1426,C 0.1455,E1 2.9895,E2 282.8128} C_DIS
LIN {X -135.655,Y 26.7663,Z 185,A 172.0432,B 3.1424,C 0.1485,E1 2.9886,E2 281.2136} C_DIS
LIN {X -136.3393,Y 23.0153,Z 185,A 173.4925,B 3.1422,C 0.1534,E1 2.9879,E2 279.782} C_DIS
LIN {X -136.8342,Y 19.8635,Z 185,A 174.9281,B 3.142,C 0.1566,E1 2.9873,E2 278.3329} C_DIS
LIN {X -137.2,Y 17.1717,Z 185,A 176.2515,B 3.142,C 0.159,E1 2.9869,E2 276.9851} C_DIS
LIN {X -137.6065,Y 13.5135,Z 185,A 177.7014,B 3.1417,C 0.1636,E1 2.9864,E2 275.5458} C_DIS
LIN {X -137.8953,Y 10.148,Z 185,A 179.119,B 3.1415,C 0.1674,E1 2.9861,E2 274.127} C_DIS
LIN {X -138.133,Y 6.1641,Z 185,A -178.9636,B 3.1413,C 0.1711,E1 2.9858,E2 272.1769} C_DIS
LIN {X -138.2364,Y 3.069,Z 185,A -177.7625,B 3.1411,C 0.175,E1 2.9858,E2 270.9872} C_DIS
LIN {X -138.2715,Y 0,Z 185,A -176.2626,B 3.1409,C 0.1777,E1 2.9858,E2 269.4589} C_DIS
LIN {X -138.2161,Y -3.7968,Z 185,A -174.793,B 3.1406,C 0.1825,E1 2.9858,E2 268.0036} C_DIS
LIN {X -138.0547,Y -7.7208,Z 185,A -173.0698,B 3.1404,C 0.1867,E1 2.9861,E2 266.2691} C_DIS
LIN {X -137.8186,Y -11.1511,Z 185,A -171.6911,B 3.1401,C 0.1909,E1 2.9863,E2 264.8972} C_DIS
LIN {X -137.5596,Y -14.0022,Z 185,A -170.1826,B 3.1401,C 0.193,E1 2.9868,E2 263.3479} C_DIS
LIN {X -137.1664,Y -17.4281,Z 185,A -168.7604,B 3.1398,C 0.197,E1 2.9872,E2 261.9273} C_DIS
LIN {X -136.687,Y -20.8522,Z 185,A -167.5204,B 3.1395,C 0.2017,E1 2.9877,E2 260.713} C_DIS
LIN {X -136.2491,Y -23.5563,Z 185,A -165.9862,B 3.1394,C 0.2033,E1 2.9885,E2 259.1279} C_DIS
LIN {X -135.5537,Y -27.2643,Z 185,A -164.4961,B 3.1391,C 0.2079,E1 2.9893,E2 257.6481} C_DIS
LIN {X -134.8662,Y -30.4833,Z 185,A -163.0598,B 3.1388,C 0.2113,E1 2.9901,E2 256.2031} C_DIS
LIN {X -134.0772,Y -33.7842,Z 185,A -161.6132,B 3.1386,C 0.215,E1 2.9911,E2 254.752} C_DIS
LIN {X -133.2212,Y -37.016,Z 185,A -160.142,B 3.1383,C 0.2184,E1 2.9922,E2 253.2704} C_DIS
LIN {X -132.2855,Y -40.2318,Z 185,A -158.7085,B 3.1381,C 0.2219,E1 2.9933,E2 251.8317} C_DIS
LIN {X -131.4535,Y -42.88,Z 185,A -157.4854,B 3.1379,C 0.2247,E1 2.9944,E2 250.5997} C_DIS
LIN {X -130.361,Y -46.0946,Z 185,A -156.0136,B 3.1377,C 0.2281,E1 2.9957,E2 249.1201} C_DIS
LIN {X -129.1832,Y -49.2991,Z 185,A -154.5342,B 3.1374,C 0.2315,E1 2.9972,E2 247.6329} C_DIS
LIN {X -127.8003,Y -52.7765,Z 185,A -152.8513,B 3.1372,C 0.235,E1 2.999,E2 245.9332} C_DIS
LIN {X -126.3518,Y -56.1543,Z 185,A -151.3233,B 3.1369,C 0.2388,E1 3.0007,E2 244.4052} C_DIS
LIN {X -124.8913,Y -59.3315,Z 185,A -149.8164,B 3.1366,C 0.2422,E1 3.0025,E2 242.8913} C_DIS
LIN {X -123.3702,Y -62.4328,Z 185,A -148.3184,B 3.1363,C 0.2454,E1 3.0044,E2 241.3851} C_DIS
LIN {X -121.5956,Y -65.8272,Z 185,A -146.5351,B 3.1361,C 0.2484,E1 3.0067,E2 239.5766} C_DIS
LIN {X -119.444,Y -69.6551,Z 185,A -144.701,B 3.1358,C 0.2527,E1 3.0093,E2 237.7412} C_DIS
LIN {X -117.1623,Y -73.4282,Z 185,A -142.8012,B 3.1354,C 0.2567,E1 3.0121,E2 235.8325} C_DIS
LIN {X -114.905,Y -76.9115,Z 185,A -141.039,B 3.1351,C 0.2604,E1 3.0148,E2 234.0651} C_DIS
LIN {X -112.3774,Y -80.5597,Z 185,A -139.1353,B 3.1348,C 0.2642,E1 3.0179,E2 232.1534} C_DIS
LIN {X -109.9329,Y -83.8648,Z 185,A -137.3109,B 3.1346,C 0.2674,E1 3.021,E2 230.3134} C_DIS
LIN {X -107.168,Y -87.3703,Z 185,A -135.3979,B 3.1342,C 0.271,E1 3.0243,E2 228.3924} C_DIS
LIN {X -104.2944,Y -90.7812,Z 185,A -133.5114,B 3.1339,C 0.2746,E1 3.0278,E2 226.5013} C_DIS
LIN {X -101.4515,Y -93.9482,Z 185,A -131.6383,B 3.1337,C 0.2776,E1 3.0313,E2 224.6138} C_DIS
LIN {X -98.4027,Y -97.1371,Z 185,A -129.7978,B 3.1334,C 0.281,E1 3.0349,E2 222.7719} C_DIS
LIN {X -95.4088,Y -100.0785,Z 185,A -128.0359,B 3.1331,C 0.2841,E1 3.0384,E2 221.0073} C_DIS
LIN {X -92.2019,Y -103.0404,Z 185,A -126.1543,B 3.1328,C 0.287,E1 3.0424,E2 219.1161} C_DIS
LIN {X -89.2148,Y -105.6382,Z 185,A -124.4545,B 3.1326,C 0.2895,E1 3.046,E2 217.4086} C_DIS
LIN {X -85.7817,Y -108.4444,Z 185,A -122.592,B 3.1323,C 0.2924,E1 3.05,E2 215.5428} C_DIS
LIN {X -82.7136,Y -110.8016,Z 185,A -120.9899,B 3.1321,C 0.295,E1 3.0536,E2 213.9408} C_DIS
LIN {X -79.5594,Y -113.0877,Z 185,A -119.262,B 3.1319,C 0.2968,E1 3.0576,E2 212.1977} C_DIS
LIN {X -75.7394,Y -115.6814,Z 185,A -117.3009,B 3.1317,C 0.2993,E1 3.0622,E2 210.2302} C_DIS
LIN {X -71.926,Y -118.0905,Z 185,A -115.4013,B 3.1315,C 0.3016,E1 3.0667,E2 208.3264} C_DIS
LIN {X -68.1302,Y -120.3204,Z 185,A -113.4765,B 3.1313,C 0.3034,E1 3.0714,E2 206.388} C_DIS
LIN {X -65.0556,Y -122.0101,Z 185,A -112.1247,B 3.1311,C 0.3057,E1 3.0747,E2 205.0497} C_DIS
LIN {X -61.951,Y -123.6155,Z 185,A -110.6505,B 3.1309,C 0.3072,E1 3.0783,E2 203.5718} C_DIS
LIN {X -58.4822,Y -125.2918,Z 185,A -109.0692,B 3.1307,C 0.309,E1 3.0823,E2 201.9924} C_DIS
LIN {X -55.665,Y -126.5706,Z 185,A -107.7257,B 3.1307,C 0.3099,E1 3.0858,E2 200.6404} C_DIS
LIN {X -52.0719,Y -128.0885,Z 185,A -106.2537,B 3.1304,C 0.3123,E1 3.0895,E2 199.1875} C_DIS
LIN {X -49.0586,Y -129.2733,Z 185,A -104.6537,B 3.1304,C 0.3118,E1 3.0938,E2 197.5525} C_DIS
LIN {X -45.5971,Y -130.5335,Z 185,A -103.1834,B 3.1303,C 0.3134,E1 3.0977,E2 196.0894} C_DIS
LIN {X -42.88,Y -131.4535,Z 185,A -101.9394,B 3.1303,C 0.3139,E1 3.101,E2 194.8378} C_DIS
LIN {X -39.1356,Y -132.6141,Z 185,A -100.351,B 3.1301,C 0.3152,E1 3.1052,E2 193.2537} C_DIS
LIN {X -36.3271,Y -133.4125,Z 185,A -99.1624,B 3.1301,C 0.3161,E1 3.1084,E2 192.0677} C_DIS
LIN {X -33.2077,Y -134.2236,Z 185,A -97.7765,B 3.13,C 0.3165,E1 3.1122,E2 190.6747} C_DIS
LIN {X -29.9843,Y -134.9802,Z 185,A -96.3964,B 3.13,C 0.317,E1 3.1159,E2 189.293} C_DIS
LIN {X -26.2371,Y -135.7562,Z 185,A -94.8116,B 3.1299,C 0.3177,E1 3.1203,E2 187.7077} C_DIS
LIN {X -23.0605,Y -136.3318,Z 185,A -93.6448,B 3.1297,C 0.3193,E1 3.1234,E2 186.5635} C_DIS
LIN {X -19.8635,Y -136.8342,Z 185,A -92.1167,B 3.1297,C 0.3183,E1 3.1277,E2 185.0097} C_DIS
LIN {X -17.1717,Y -137.2,Z 185,A -90.8511,B 3.1299,C 0.3175,E1 3.1313,E2 183.7248} C_DIS
LIN {X -13.4215,Y -137.6154,Z 185,A -89.4434,B 3.1297,C 0.3189,E1 3.1352,E2 182.3375} C_DIS
LIN {X -10.3656,Y -137.8794,Z 185,A -88.1555,B 3.1297,C 0.3189,E1 3.1388,E2 181.0468} C_DIS
LIN {X -6.1641,Y -138.133,Z 185,A -86.2813,B 3.1299,C 0.3178,E1 3.144,E2 179.1543} C_DIS
LIN {X -3.069,Y -138.2364,Z 185,A -84.9932,B 3.1299,C 0.3177,E1 3.1477,E2 177.865} C_DIS
LIN {X 0.9813,Y -138.2634,Z 185,A -83.5476,B 3.1297,C 0.3191,E1 3.1516,E2 176.45} C_DIS
Enddeposition()
LIN {X 0.9813,Y -138.2634,Z 185,A -83.5476,B 3.1297,C 0.3191,E1 3.1516,E2 176.45} C_DIS
Startdeposition()
$VEL.CP = VEL_PRINT
LIN {X -0.8684,Y -139.1658,Z 185,A -84.8355,B 3.1381,C 0.3252,E1 3.1567,E2 177.8376} C_DIS
LIN {X -5.2673,Y -139.0688,Z 185,A -86.6266,B 3.1381,C 0.3252,E1 3.1517,E2 179.6267} C_DIS
LIN {X -9.0765,Y -138.8731,Z 185,A -88.3052,B 3.138,C 0.326,E1 3.147,E2 181.3207} C_DIS
LIN {X -13.3217,Y -138.5293,Z 185,A -89.9336,B 3.1381,C 0.325,E1 3.1425,E2 182.933} C_DIS
LIN {X -16.6889,Y -138.1642,Z 185,A -91.3755,B 3.1381,C 0.3251,E1 3.1384,E2 184.3818} C_DIS
LIN {X -21.1703,Y -137.5487,Z 185,A -93.2817,B 3.1381,C 0.325,E1 3.1331,E2 186.2946} C_DIS
LIN {X -26.4417,Y -136.6335,Z 185,A -95.464,B 3.1381,C 0.3241,E1 3.1271,E2 188.4749} C_DIS
LIN {X -34.5169,Y -134.82,Z 185,A -98.8896,B 3.1383,C 0.3226,E1 3.1178,E2 191.9041} C_DIS
LIN {X -37.8413,Y -133.9251,Z 185,A -100.2699,B 3.1385,C 0.3215,E1 3.1141,E2 193.2798} C_DIS
LIN {X -41.0405,Y -132.9794,Z 185,A -101.7065,B 3.1385,C 0.321,E1 3.1102,E2 194.7252} C_DIS
LIN {X -45.4775,Y -131.5277,Z 185,A -103.8655,B 3.1385,C 0.3211,E1 3.1044,E2 196.9165} C_DIS
LIN {X -50.6582,Y -129.6207,Z 185,A -105.9292,B 3.1388,C 0.3179,E1 3.0991,E2 198.9526} C_DIS
LIN {X -54.31,Y -128.1354,Z 185,A -107.5631,B 3.139,C 0.3165,E1 3.0949,E2 200.5883} C_DIS
LIN {X -58.4745,Y -126.2871,Z 185,A -109.4138,B 3.1392,C 0.3144,E1 3.0902,E2 202.4359} C_DIS
LIN {X -66.6678,Y -122.1625,Z 185,A -113.4026,B 3.1395,C 0.3114,E1 3.0802,E2 206.4538} C_DIS
LIN {X -70.6338,Y -119.9131,Z 185,A -115.3295,B 3.1397,C 0.3093,E1 3.0755,E2 208.3875} C_DIS
LIN {X -74.5818,Y -117.4987,Z 185,A -117.3448,B 3.1399,C 0.3073,E1 3.0707,E2 210.4176} C_DIS
LIN {X -77.7836,Y -115.4038,Z 185,A -120.0405,B 3.1395,C 0.3113,E1 3.0642,E2 213.2617} C_DIS
LIN {X -84.5845,Y -110.5157,Z 185,A -122.4152,B 3.1406,C 0.3,E1 3.0591,E2 215.4945} C_DIS
LIN {X -88.154,Y -107.69,Z 185,A -124.3506,B 3.1409,C 0.2972,E1 3.0549,E2 217.438} C_DIS
LIN {X -91.8205,Y -104.5822,Z 185,A -126.3903,B 3.1411,C 0.2941,E1 3.0505,E2 219.4856} C_DIS
LIN {X -95.1408,Y -101.5709,Z 185,A -128.3065,B 3.1414,C 0.2912,E1 3.0466,E2 221.411} C_DIS
LIN {X -99.2917,Y -97.5163,Z 185,A -130.7034,B 3.1418,C 0.2867,E1 3.0418,E2 223.8087} C_DIS
LIN {X -102.2112,Y -94.4524,Z 185,A -132.6354,B 3.1421,C 0.2842,E1 3.0381,E2 225.7655} C_DIS
LIN {X -105.0854,Y -91.2438,Z 185,A -134.3537,B 3.1424,C 0.2804,E1 3.0349,E2 227.4762} C_DIS
LIN {X -107.9397,Y -87.8485,Z 185,A -136.2455,B 3.1427,C 0.2769,E1 3.0315,E2 229.3763} C_DIS
LIN {X -110.5683,Y -84.5157,Z 185,A -138.4503,B 3.1428,C 0.2753,E1 3.0277,E2 231.6408} C_DIS
LIN {X -113.0442,Y -81.1748,Z 185,A -139.5623,B 3.1434,C 0.2687,E1 3.026,E2 232.6733} C_DIS
LIN {X -114.8033,Y -78.6668,Z 185,A -141.1567,B 3.1435,C 0.2674,E1 3.0234,E2 234.3114} C_DIS
LIN {X -117.3107,Y -74.8765,Z 185,A -143.238,B 3.1438,C 0.2641,E1 3.0201,E2 236.4198} C_DIS
LIN {X -119.9725,Y -70.5327,Z 185,A -145.9106,B 3.144,C 0.2617,E1 3.0162,E2 239.1668} C_DIS
LIN {X -122.6446,Y -65.7768,Z 185,A -147.5689,B 3.1447,C 0.2536,E1 3.0141,E2 240.7477} C_DIS
LIN {X -124.239,Y -62.7103,Z 185,A -149.0124,B 3.1449,C 0.2502,E1 3.0123,E2 242.1932} C_DIS
LIN {X -125.746,Y -59.6305,Z 185,A -150.5081,B 3.1452,C 0.2471,E1 3.0105,E2 243.6994} C_DIS
LIN {X -127.4889,Y -55.8093,Z 185,A -152.5054,B 3.1454,C 0.2438,E1 3.0081,E2 245.731} C_DIS
LIN {X -129.2544,Y -51.5872,Z 185,A -154.2317,B 3.1459,C 0.2383,E1 3.0063,E2 247.4359} C_DIS
LIN {X -131.2369,Y -46.3164,Z 185,A -156.6473,B 3.1463,C 0.2327,E1 3.004,E2 249.8632} C_DIS
LIN {X -132.2755,Y -43.2606,Z 185,A -158.0552,B 3.1465,C 0.2295,E1 3.0027,E2 251.2808} C_DIS
LIN {X -133.1154,Y -40.596,Z 185,A -159.2847,B 3.1467,C 0.2267,E1 3.0017,E2 252.52} C_DIS
LIN {X -134.1268,Y -37.1199,Z 185,A -160.8009,B 3.147,C 0.2228,E1 3.0005,E2 254.0387} C_DIS
LIN {X -134.9084,Y -34.1687,Z 185,A -162.1679,B 3.1472,C 0.2199,E1 2.9996,E2 255.4194} C_DIS
LIN {X -135.8352,Y -30.2834,Z 185,A -164.0086,B 3.1475,C 0.2162,E1 2.9984,E2 257.2847} C_DIS
LIN {X -136.7528,Y -25.8179,Z 185,A -165.8748,B 3.1478,C 0.211,E1 2.9974,E2 259.1483} C_DIS
LIN {X -137.5734,Y -21.0105,Z 185,A -167.8799,B 3.1482,C 0.2054,E1 2.9965,E2 261.1519} C_DIS
LIN {X -138.0068,Y -17.9431,Z 185,A -169.2422,B 3.1484,C 0.2022,E1 2.996,E2 262.5248} C_DIS
LIN {X -138.399,Y -14.6156,Z 185,A -171.0083,B 3.1485,C 0.1999,E1 2.9954,E2 264.3398} C_DIS
LIN {X -138.7049,Y -11.3537,Z 185,A -172.2595,B 3.1488,C 0.1957,E1 2.9951,E2 265.5776} C_DIS
LIN {X -139.0951,Y -4.5711,Z 185,A -174.9972,B 3.1493,C 0.1876,E1 2.9948,E2 268.3059} C_DIS
LIN {X -139.1461,Y 2.5044,Z 185,A -178.1189,B 3.1497,C 0.1802,E1 2.9948,E2 271.4525} C_DIS
LIN {X -138.8748,Y 9.0475,Z 185,A 179.168,B 3.1501,C 0.1727,E1 2.9951,E2 274.166} C_DIS
LIN {X -138.6662,Y 11.812,Z 185,A 177.8895,B 3.1503,C 0.17,E1 2.9954,E2 275.4612} C_DIS
LIN {X -138.2818,Y 15.7029,Z 185,A 175.7202,B 3.1504,C 0.1677,E1 2.9961,E2 277.7005} C_DIS
LIN {X -137.776,Y 19.6362,Z 185,A 174.411,B 3.1507,C 0.1618,E1 2.9965,E2 278.9675} C_DIS
LIN {X -137.2831,Y 22.8289,Z 185,A 173.0753,B 3.1509,C 0.1582,E1 2.9971,E2 280.3031} C_DIS
LIN {X -136.6722,Y 26.2392,Z 185,A 171.4834,B 3.1511,C 0.1549,E1 2.998,E2 281.9149} C_DIS
LIN {X -135.9321,Y 29.8406,Z 185,A 169.9418,B 3.1513,C 0.1508,E1 2.9989,E2 283.459} C_DIS
LIN {X -134.8506,Y 34.3961,Z 185,A 167.98,B 3.1515,C 0.1457,E1 3.0002,E2 285.4237} C_DIS
LIN {X -133.9585,Y 37.7217,Z 185,A 166.5161,B 3.1517,C 0.142,E1 3.0012,E2 286.8924} C_DIS
LIN {X -133.0164,Y 40.9196,Z 185,A 165.0633,B 3.1518,C 0.1386,E1 3.0024,E2 288.3543} C_DIS
LIN {X -131.9356,Y 44.2813,Z 185,A 163.5155,B 3.152,C 0.1351,E1 3.0038,E2 289.9128} C_DIS
LIN {X -130.8306,Y 47.4461,Z 185,A 162.1103,B 3.1521,C 0.1315,E1 3.0051,E2 291.3201} C_DIS
LIN {X -129.5989,Y 50.7142,Z 185,A 160.602,B 3.1523,C 0.1281,E1 3.0066,E2 292.8362} C_DIS
LIN {X -128.3022,Y 53.9105,Z 185,A 159.0876,B 3.1524,C 0.1248,E1 3.0082,E2 294.3613} C_DIS
LIN {X -126.965,Y 56.9879,Z 185,A 157.72,B 3.1525,C 0.1212,E1 3.0098,E2 295.7261} C_DIS
LIN {X -125.4387,Y 60.2737,Z 185,A 156.104,B 3.1527,C 0.1179,E1 3.0117,E2 297.3566} C_DIS
LIN {X -123.7849,Y 63.6023,Z 185,A 154.5314,B 3.1528,C 0.1142,E1 3.0137,E2 298.9333} C_DIS
LIN {X -122.2765,Y 66.4587,Z 185,A 153.0318,B 3.1528,C 0.1117,E1 3.0157,E2 300.4531} C_DIS
LIN {X -119.2084,Y 71.8169,Z 185,A 150.4047,B 3.1531,C 0.1059,E1 3.0194,E2 303.0889} C_DIS
LIN {X -115.3558,Y 77.8545,Z 185,A 147.005,B 3.1533,C 0.1009,E1 3.0247,E2 306.5422} C_DIS
LIN {X -113.0983,Y 81.0992,Z 185,A 145.6936,B 3.1534,C 0.0959,E1 3.0268,E2 307.8132} C_DIS
LIN {X -110.6587,Y 84.3975,Z 185,A 143.8739,B 3.1535,C 0.0927,E1 3.0298,E2 309.6479} C_DIS
LIN {X -107.7585,Y 88.0702,Z 185,A 141.9032,B 3.1536,C 0.0888,E1 3.0333,E2 311.6225} C_DIS
LIN {X -104.8737,Y 91.4864,Z 185,A 139.6731,B 3.1536,C 0.0867,E1 3.0374,E2 313.8993} C_DIS
LIN {X -102.2561,Y 94.4036,Z 185,A 138.3203,B 3.1538,C 0.0822,E1 3.0399,E2 315.2187} C_DIS
LIN {X -99.0609,Y 97.7515,Z 185,A 136.3549,B 3.1538,C 0.0787,E1 3.0438,E2 317.1901} C_DIS
LIN {X -95.9844,Y 100.7735,Z 185,A 134.0355,B 3.1539,C 0.0779,E1 3.0486,E2 319.5749} C_DIS
LIN {X -92.4476,Y 104.028,Z 185,A 132.7677,B 3.1541,C 0.0709,E1 3.051,E2 320.7539} C_DIS
LIN {X -88.7619,Y 107.1895,Z 185,A 130.3958,B 3.1541,C 0.0692,E1 3.0562,E2 323.1703} C_DIS
LIN {X -85.9444,Y 109.4615,Z 185,A 128.1537,B 3.1541,C 0.0704,E1 3.0613,E2 325.503} C_DIS
LIN {X -81.0325,Y 113.146,Z 185,A 126.5379,B 3.1543,C 0.0619,E1 3.0647,E2 327.0057} C_DIS
LIN {X -78.3523,Y 115.0189,Z 185,A 124.9023,B 3.1543,C 0.0613,E1 3.0685,E2 328.676} C_DIS
LIN {X -75.4252,Y 116.9593,Z 185,A 123.4352,B 3.1543,C 0.0593,E1 3.072,E2 330.1448} C_DIS
LIN {X -71.7166,Y 119.2691,Z 185,A 121.4514,B 3.1543,C 0.0578,E1 3.0768,E2 332.1499} C_DIS
LIN {X -68.0835,Y 121.3792,Z 185,A 119.8332,B 3.1543,C 0.0549,E1 3.0807,E2 333.7533} C_DIS
LIN {X -63.8708,Y 123.6483,Z 185,A 117.6588,B 3.1544,C 0.0536,E1 3.0861,E2 335.9513} C_DIS
LIN {X -59.5211,Y 125.7983,Z 185,A 115.8797,B 3.1544,C 0.0501,E1 3.0905,E2 337.7023} C_DIS
LIN {X -56.7476,Y 127.0725,Z 185,A 114.5322,B 3.1544,C 0.0493,E1 3.094,E2 339.0601} C_DIS
LIN {X -52.8767,Y 128.734,Z 185,A 112.7918,B 3.1545,C 0.0476,E1 3.0984,E2 340.8003} C_DIS
LIN {X -48.2258,Y 130.5465,Z 185,A 110.476,B 3.1545,C 0.0473,E1 3.1046,E2 343.1466} C_DIS
LIN {X -43.7448,Y 132.1143,Z 185,A 108.7654,B 3.1545,C 0.0443,E1 3.109,E2 344.8262} C_DIS
LIN {X -39.8954,Y 133.3296,Z 185,A 107.0704,B 3.1545,C 0.0433,E1 3.1136,E2 346.5244} C_DIS
LIN {X -36.5659,Y 134.2804,Z 185,A 105.6958,B 3.1545,C 0.0421,E1 3.1172,E2 347.8919} C_DIS
LIN {X -32.244,Y 135.3818,Z 185,A 103.6823,B 3.1545,C 0.0421,E1 3.1228,E2 349.926} C_DIS
LIN {X -27.7722,Y 136.3689,Z 185,A 101.8505,B 3.1546,C 0.0409,E1 3.1277,E2 351.7501} C_DIS
LIN {X -23.488,Y 137.1731,Z 185,A 99.9805,B 3.1546,C 0.0407,E1 3.1329,E2 353.6284} C_DIS
LIN {X -18.8631,Y 137.8862,Z 185,A 98.1804,B 3.1546,C 0.0393,E1 3.1378,E2 355.4122} C_DIS
LIN {X -15.5825,Y 138.2949,Z 185,A 96.5487,B 3.1546,C 0.0408,E1 3.1425,E2 357.0762} C_DIS
LIN {X -10.253,Y 138.7902,Z 185,A 94.1931,B 3.1546,C 0.0415,E1 3.1491,E2 359.4491} C_DIS
LIN {X -6.3321,Y 139.0258,Z 185,A 92.982,B 3.1546,C 0.0388,E1 3.1523,E2 360.6101} C_DIS
LIN {X -2.5362,Y 139.1455,Z 185,A 91.3852,B 3.1546,C 0.039,E1 3.1568,E2 362.2103} C_DIS
LIN {X 1.072,Y 139.1647,Z 185,A 89.911,B 3.1546,C 0.0391,E1 3.1609,E2 363.6824} C_DIS
LIN {X 5.1877,Y 139.0719,Z 185,A 88.1719,B 3.1546,C 0.0398,E1 3.1658,E2 365.4263} C_DIS
LIN {X 8.6303,Y 138.9005,Z 185,A 86.821,B 3.1546,C 0.0398,E1 3.1695,E2 366.7683} C_DIS
LIN {X 12.3805,Y 138.6182,Z 185,A 85.1495,B 3.1546,C 0.0411,E1 3.1742,E2 368.4543} C_DIS
LIN {X 16.4542,Y 138.1922,Z 185,A 83.6104,B 3.1546,C 0.0408,E1 3.1785,E2 369.9748} C_DIS
LIN {X 23.1424,Y 137.2308,Z 185,A 81.0281,B 3.1546,C 0.0408,E1 3.1855,E2 372.5318} C_DIS
LIN {X 31.4881,Y 135.56,Z 185,A 77.3563,B 3.1546,C 0.0445,E1 3.1957,E2 376.2233} C_DIS
LIN {X 35.8228,Y 134.4785,Z 185,A 75.5666,B 3.1546,C 0.0455,E1 3.2005,E2 378.0066} C_DIS
LIN {X 39.1592,Y 133.5451,Z 185,A 74.0543,B 3.1546,C 0.0475,E1 3.2046,E2 379.529} C_DIS
LIN {X 42.3892,Y 132.5552,Z 185,A 72.5656,B 3.1545,C 0.0496,E1 3.2086,E2 381.0294} C_DIS
LIN {X 47.7103,Y 130.7354,Z 185,A 70.5145,B 3.1545,C 0.0499,E1 3.2139,E2 383.0478} C_DIS
LIN {X 51.1503,Y 129.4294,Z 185,A 69.0183,B 3.1545,C 0.0514,E1 3.2178,E2 384.5414} C_DIS
LIN {X 54.2576,Y 128.1573,Z 185,A 67.5495,B 3.1545,C 0.0537,E1 3.2216,E2 386.0206} C_DIS
LIN {X 58.4669,Y 126.2907,Z 185,A 65.1122,B 3.1543,C 0.0606,E1 3.228,E2 388.5238} C_DIS
LIN {X 63.4978,Y 123.8381,Z 185,A 63.4777,B 3.1543,C 0.0582,E1 3.2318,E2 390.0762} C_DIS
LIN {X 67.6603,Y 121.6159,Z 185,A 61.5494,B 3.1543,C 0.0608,E1 3.2366,E2 392.0026} C_DIS
LIN {X 71.6124,Y 119.3319,Z 185,A 59.75,B 3.1543,C 0.063,E1 3.2409,E2 393.7921} C_DIS
LIN {X 75.0382,Y 117.2072,Z 185,A 58.0683,B 3.1542,C 0.0658,E1 3.2448,E2 395.4765} C_DIS
LIN {X 81.5724,Y 112.7573,Z 185,A 55.0684,B 3.1542,C 0.0691,E1 3.2517,E2 398.445} C_DIS
LIN {X 84.7358,Y 110.4,Z 185,A 53.367,B 3.154,C 0.0726,E1 3.2555,E2 400.1559} C_DIS
LIN {X 88.2128,Y 107.642,Z 185,A 51.4904,B 3.154,C 0.0764,E1 3.2596,E2 402.0388} C_DIS
LIN {X 92.0075,Y 104.4171,Z 185,A 48.8807,B 3.1537,C 0.0854,E1 3.2652,E2 404.7177} C_DIS
LIN {X 96.6028,Y 100.1809,Z 185,A 47.0993,B 3.1537,C 0.0834,E1 3.2686,E2 406.4017} C_DIS
LIN {X 99.7543,Y 97.0435,Z 185,A 45.3071,B 3.1537,C 0.0868,E1 3.2721,E2 408.1894} C_DIS
LIN {X 102.8676,Y 93.7369,Z 185,A 43.3359,B 3.1535,C 0.0917,E1 3.2759,E2 410.1735} C_DIS
LIN {X 105.0311,Y 91.3061,Z 185,A 42.4717,B 3.1535,C 0.0902,E1 3.2774,E2 410.9786} C_DIS
LIN {X 110.2374,Y 84.9478,Z 185,A 39.1134,B 3.1534,C 0.0975,E1 3.2833,E2 414.3347} C_DIS
LIN {X 112.4172,Y 82.0415,Z 185,A 37.4798,B 3.1532,C 0.1022,E1 3.286,E2 415.986} C_DIS
LIN {X 115.0257,Y 78.3423,Z 185,A 35.6837,B 3.1531,C 0.106,E1 3.2889,E2 417.7742} C_DIS
LIN {X 117.5437,Y 74.5105,Z 185,A 33.8762,B 3.153,C 0.1097,E1 3.2916,E2 419.5722} C_DIS
LIN {X 119.9689,Y 70.5388,Z 185,A 32.0563,B 3.1528,C 0.1135,E1 3.2942,E2 421.3806} C_DIS
LIN {X 122.1682,Y 66.6574,Z 185,A 30.2954,B 3.1527,C 0.1173,E1 3.2966,E2 423.1326} C_DIS
LIN {X 123.9191,Y 63.3387,Z 185,A 28.8564,B 3.1526,C 0.1202,E1 3.2984,E2 424.5588} C_DIS
LIN {X 125.7361,Y 59.6513,Z 185,A 27.2798,B 3.1525,C 0.1234,E1 3.3003,E2 426.1214} C_DIS
LIN {X 127.1329,Y 56.6125,Z 185,A 25.9536,B 3.1523,C 0.1264,E1 3.3018,E2 427.4417} C_DIS
LIN {X 128.501,Y 53.4345,Z 185,A 24.5856,B 3.1523,C 0.1296,E1 3.3033,E2 428.8031} C_DIS
LIN {X 130.0193,Y 49.6327,Z 185,A 22.9453,B 3.152,C 0.1336,E1 3.305,E2 430.4385} C_DIS
LIN {X 131.1027,Y 46.6916,Z 185,A 21.7652,B 3.152,C 0.1359,E1 3.3061,E2 431.6051} C_DIS
LIN {X 132.1077,Y 43.7646,Z 185,A 20.4879,B 3.1518,C 0.1394,E1 3.3072,E2 432.8834} C_DIS
LIN {X 133.2377,Y 40.1967,Z 185,A 18.9358,B 3.1516,C 0.1436,E1 3.3085,E2 434.4377} C_DIS
LIN {X 134.5032,Y 35.7304,Z 185,A 17.2474,B 3.1515,C 0.1466,E1 3.3098,E2 436.0986} C_DIS
LIN {X 135.2996,Y 32.585,Z 185,A 15.9094,B 3.1513,C 0.1503,E1 3.3107,E2 437.4376} C_DIS
LIN {X 136.1316,Y 28.9167,Z 185,A 14.4935,B 3.1512,C 0.1532,E1 3.3115,E2 438.8374} C_DIS
LIN {X 136.6741,Y 26.2295,Z 185,A 12.7226,B 3.1507,C 0.1628,E1 3.3125,E2 440.6908} C_DIS
LIN {X 137.5854,Y 20.9328,Z 185,A 11.2955,B 3.1507,C 0.161,E1 3.3131,E2 442.0189} C_DIS
LIN {X 138.0262,Y 17.7953,Z 185,A 9.9538,B 3.1506,C 0.1651,E1 3.3136,E2 443.3661} C_DIS
LIN {X 138.5146,Y 13.4749,Z 185,A 8.2478,B 3.1503,C 0.1692,E1 3.3141,E2 445.0624} C_DIS
LIN {X 138.8294,Y 9.7162,Z 185,A 6.804,B 3.1502,C 0.1725,E1 3.3144,E2 446.493} C_DIS
LIN {X 139.0512,Y 5.7185,Z 185,A 5.1759,B 3.1499,C 0.1769,E1 3.3146,E2 448.1196} C_DIS
LIN {X 139.1613,Y 1.5877,Z 185,A 3.4645,B 3.1496,C 0.1818,E1 3.3146,E2 449.8335} C_DIS
LIN {X 139.1458,Y -2.5185,Z 185,A 1.9005,B 3.1494,C 0.1853,E1 3.3146,E2 451.3822} C_DIS
LIN {X 138.9988,Y -6.8703,Z 185,A 0.2413,B 3.1492,C 0.189,E1 3.3144,E2 453.0252} C_DIS
LIN {X 138.788,Y -10.2834,Z 185,A -1.0956,B 3.149,C 0.1922,E1 3.3142,E2 454.3538} C_DIS
LIN {X 138.4607,Y -14.0363,Z 185,A -2.7196,B 3.1487,C 0.1973,E1 3.3138,E2 455.9886} C_DIS
LIN {X 137.9392,Y -18.4587,Z 185,A -4.2801,B 3.1486,C 0.1997,E1 3.3132,E2 457.5148} C_DIS
LIN {X 137.2091,Y -23.2723,Z 185,A -6.3018,B 3.1482,C 0.2054,E1 3.3124,E2 459.5402} C_DIS
LIN {X 135.7252,Y -30.7652,Z 185,A -9.0469,B 3.1479,C 0.2101,E1 3.3109,E2 462.2353} C_DIS
LIN {X 134.3872,Y -36.1654,Z 185,A -11.3581,B 3.1474,C 0.2166,E1 3.3093,E2 464.5511} C_DIS
LIN {X 133.5902,Y -39.0054,Z 185,A -12.6698,B 3.1471,C 0.2209,E1 3.3083,E2 465.8765} C_DIS
LIN {X 132.5089,Y -42.5344,Z 185,A -14.1395,B 3.1469,C 0.2245,E1 3.3071,E2 467.3408} C_DIS
LIN {X 131.356,Y -45.9729,Z 185,A -15.8547,B 3.1464,C 0.2308,E1 3.3055,E2 469.0863} C_DIS
LIN {X 130.0446,Y -49.5658,Z 185,A -17.0121,B 3.1464,C 0.2308,E1 3.3044,E2 470.1902} C_DIS
LIN {X 129.0006,Y -52.2169,Z 185,A -18.1666,B 3.1462,C 0.2336,E1 3.3032,E2 471.3431} C_DIS
LIN {X 127.2894,Y -56.2627,Z 185,A -20.0983,B 3.1458,C 0.2396,E1 3.301,E2 473.2925} C_DIS
LIN {X 125.4548,Y -60.24,Z 185,A -21.6413,B 3.1456,C 0.2416,E1 3.2992,E2 474.8026} C_DIS
LIN {X 123.5787,Y -64.0048,Z 185,A -23.2508,B 3.1454,C 0.2448,E1 3.2972,E2 476.3973} C_DIS
LIN {X 121.9001,Y -67.147,Z 185,A -25.1102,B 3.1448,C 0.2525,E1 3.2946,E2 478.3097} C_DIS
LIN {X 119.8429,Y -70.7533,Z 185,A -26.2498,B 3.1448,C 0.251,E1 3.2931,E2 479.3755} C_DIS
LIN {X 117.9753,Y -73.8255,Z 185,A -27.8513,B 3.1445,C 0.2558,E1 3.2908,E2 480.9943} C_DIS
LIN {X 115.3418,Y -77.8753,Z 185,A -29.6297,B 3.1443,C 0.2585,E1 3.2881,E2 482.7464} C_DIS
LIN {X 113.1706,Y -80.998,Z 185,A -31.6287,B 3.1436,C 0.2665,E1 3.2847,E2 484.8041} C_DIS
LIN {X 110.6132,Y -84.457,Z 185,A -32.625,B 3.1439,C 0.263,E1 3.2833,E2 485.6989} C_DIS
LIN {X 107.4347,Y -88.4658,Z 185,A -35.0426,B 3.1432,C 0.2708,E1 3.2789,E2 488.1598} C_DIS
LIN {X 103.9355,Y -92.5518,Z 185,A -37.1813,B 3.1429,C 0.2749,E1 3.275,E2 490.2902} C_DIS
LIN {X 100.869,Y -95.8845,Z 185,A -38.9549,B 3.1426,C 0.2781,E1 3.2717,E2 492.0531} C_DIS
LIN {X 97.8584,Y -98.955,Z 185,A -40.6724,B 3.1423,C 0.2812,E1 3.2683,E2 493.765} C_DIS
LIN {X 94.4528,Y -102.2106,Z 185,A -42.5686,B 3.142,C 0.2847,E1 3.2644,E2 495.657} C_DIS
LIN {X 91.4894,Y -104.8711,Z 185,A -44.1165,B 3.1418,C 0.2871,E1 3.2612,E2 497.1939} C_DIS
LIN {X 88.1405,Y -107.7011,Z 185,A -45.8786,B 3.1415,C 0.2901,E1 3.2575,E2 498.9516} C_DIS
LIN {X 83.8184,Y -111.0978,Z 185,A -48.0215,B 3.1412,C 0.2931,E1 3.2528,E2 501.0803} C_DIS
LIN {X 80.6648,Y -113.4089,Z 185,A -49.6665,B 3.1409,C 0.2963,E1 3.249,E2 502.7313} C_DIS
LIN {X 76.9456,Y -115.9644,Z 185,A -51.4153,B 3.1407,C 0.2984,E1 3.245,E2 504.4668} C_DIS
LIN {X 72.2146,Y -118.9679,Z 185,A -53.724,B 3.1404,C 0.3021,E1 3.2395,E2 506.7775} C_DIS
LIN {X 68.356,Y -121.226,Z 185,A -55.5169,B 3.1402,C 0.3045,E1 3.2352,E2 508.5653} C_DIS
LIN {X 64.4234,Y -123.3588,Z 185,A -57.2663,B 3.14,C 0.3064,E1 3.2309,E2 510.3036} C_DIS
LIN {X 60.9235,Y -125.1261,Z 185,A -58.8512,B 3.1398,C 0.3083,E1 3.2269,E2 511.8858} C_DIS
LIN {X 57.9722,Y -126.5194,Z 185,A -60.1121,B 3.1397,C 0.3094,E1 3.2238,E2 513.1364} C_DIS
LIN {X 54.8514,Y -127.9031,Z 185,A -61.4895,B 3.1395,C 0.3109,E1 3.2202,E2 514.5111} C_DIS
LIN {X 51.1873,Y -129.415,Z 185,A -63.6073,B 3.1389,C 0.3171,E1 3.2146,E2 516.6953} C_DIS
LIN {X 46.9519,Y -131.0088,Z 185,A -64.8569,B 3.1392,C 0.3139,E1 3.2115,E2 517.8637} C_DIS
LIN {X 43.7971,Y -132.0969,Z 185,A -66.2646,B 3.1391,C 0.3156,E1 3.2078,E2 519.2769} C_DIS
LIN {X 40.596,Y -133.1154,Z 185,A -67.6323,B 3.1389,C 0.3168,E1 3.2041,E2 520.6434} C_DIS
LIN {X 36.7601,Y -134.2275,Z 185,A -69.2416,B 3.1389,C 0.3181,E1 3.1998,E2 522.2491} C_DIS
LIN {X 30.9605,Y -135.6806,Z 185,A -71.6557,B 3.1386,C 0.3197,E1 3.1933,E2 524.6583} C_DIS
LIN {X 27.5429,Y -136.4156,Z 185,A -73.5362,B 3.1382,C 0.3243,E1 3.1879,E2 526.5991} C_DIS
LIN {X 23.407,Y -137.1866,Z 185,A -74.8393,B 3.1384,C 0.322,E1 3.1845,E2 527.8455} C_DIS
LIN {X 16.5158,Y -138.1848,Z 185,A -77.6101,B 3.1384,C 0.3228,E1 3.1769,E2 530.605} C_DIS
LIN {X 13.133,Y -138.5474,Z 185,A -79.0493,B 3.1382,C 0.3238,E1 3.1728,E2 532.0502} C_DIS
LIN {X 9.1231,Y -138.8702,Z 185,A -80.7869,B 3.1382,C 0.325,E1 3.168,E2 533.7996} C_DIS
LIN {X 4.9363,Y -139.0817,Z 185,A -82.3907,B 3.1382,C 0.3246,E1 3.1635,E2 535.3878} C_DIS
LIN {X 0.9816,Y -139.1651,Z 185,A -84.0591,B 3.1381,C 0.3252,E1 3.1588,E2 537.0624} C_DIS
Enddeposition()
LIN {X 0.9816,Y -139.1651,Z 185,A -84.0591,B 3.1381,C 0.3252,E1 3.1588,E2 537.0624} C_DIS
Startdeposition()
$VEL.CP = VEL_PRINT
LIN {X 1.9055,Y -140.0563,Z 185,A -82.9791,B 3.148,C 0.3218,E1 3.1716,E2 535.9145} C_DIS
LIN {X 5.6344,Y -139.9553,Z 185,A -81.4432,B 3.148,C 0.3213,E1 3.1759,E2 534.3764} C_DIS
LIN {X 9.945,Y -139.7153,Z 185,A -79.7133,B 3.148,C 0.321,E1 3.1807,E2 532.6507} C_DIS
LIN {X 13.6272,Y -139.4042,Z 185,A -78.2186,B 3.1481,C 0.3205,E1 3.1848,E2 531.1575} C_DIS
LIN {X 16.9553,Y -139.0389,Z 185,A -76.8991,B 3.1481,C 0.3202,E1 3.1885,E2 529.8441} C_DIS
LIN {X 21.4357,Y -138.4185,Z 185,A -74.9717,B 3.1483,C 0.3185,E1 3.1938,E2 527.905} C_DIS
LIN {X 28.33,Y -137.174,Z 185,A -72.0876,B 3.1485,C 0.3164,E1 3.2018,E2 525.0168} C_DIS
LIN {X 32.4668,Y -136.2541,Z 185,A -70.3715,B 3.1486,C 0.3152,E1 3.2065,E2 523.302} C_DIS
LIN {X 37.2596,Y -135.0224,Z 185,A -68.4558,B 3.1487,C 0.3144,E1 3.2116,E2 521.4} C_DIS
LIN {X 41.0345,Y -133.9226,Z 185,A -66.9326,B 3.1488,C 0.3135,E1 3.2156,E2 519.8874} C_DIS
LIN {X 44.1032,Y -132.9437,Z 185,A -65.6951,B 3.1488,C 0.3129,E1 3.2189,E2 518.6601} C_DIS
LIN {X 47.4671,Y -131.78,Z 185,A -63.9077,B 3.1493,C 0.3084,E1 3.2237,E2 516.826} C_DIS
LIN {X 50.6186,Y -130.6019,Z 185,A -62.8974,B 3.1492,C 0.3101,E1 3.2262,E2 515.8652} C_DIS
LIN {X 53.8119,Y -129.3189,Z 185,A -61.4597,B 3.1494,C 0.3081,E1 3.23,E2 514.4224} C_DIS
LIN {X 58.8569,Y -127.102,Z 185,A -59.306,B 3.1495,C 0.3061,E1 3.2355,E2 512.2809} C_DIS
LIN {X 61.6589,Y -125.767,Z 185,A -58.1946,B 3.1495,C 0.3058,E1 3.2382,E2 511.1902} C_DIS
LIN {X 65.0759,Y -124.0329,Z 185,A -56.5229,B 3.1499,C 0.3026,E1 3.2424,E2 509.5032} C_DIS
LIN {X 68.6877,Y -122.0722,Z 185,A -54.7555,B 3.1502,C 0.2993,E1 3.2467,E2 507.7228} C_DIS
LIN {X 72.0517,Y -120.118,Z 185,A -52.5663,B 3.1509,C 0.2913,E1 3.2522,E2 505.4501} C_DIS
LIN {X 76.965,Y -117.03,Z 185,A -50.8858,B 3.1507,C 0.2939,E1 3.2559,E2 503.8632} C_DIS
LIN {X 80.7695,Y -114.4374,Z 185,A -49.2167,B 3.1508,C 0.2927,E1 3.2597,E2 502.222} C_DIS
LIN {X 84.9193,Y -111.3929,Z 185,A -46.4528,B 3.1517,C 0.2826,E1 3.2661,E2 499.3662} C_DIS
LIN {X 89.1399,Y -108.0452,Z 185,A -44.86,B 3.1516,C 0.2843,E1 3.2693,E2 497.8555} C_DIS
LIN {X 92.3648,Y -105.3019,Z 185,A -42.7505,B 3.1522,C 0.2773,E1 3.2739,E2 495.6929} C_DIS
LIN {X 95.8531,Y -102.1368,Z 185,A -41.2002,B 3.1522,C 0.2771,E1 3.2769,E2 494.1927} C_DIS
LIN {X 99.625,Y -98.4612,Z 185,A -39.2195,B 3.1525,C 0.2743,E1 3.2808,E2 492.234} C_DIS
LIN {X 102.6729,Y -95.2783,Z 185,A -37.638,B 3.1526,C 0.2727,E1 3.2838,E2 490.681} C_DIS
LIN {X 106.9232,Y -90.4829,Z 185,A -34.9391,B 3.1532,C 0.2662,E1 3.2888,E2 487.9696} C_DIS
LIN {X 109.7328,Y -87.0539,Z 185,A -33.1966,B 3.1535,C 0.2628,E1 3.2918,E2 486.2352} C_DIS
LIN {X 113.6282,Y -81.9043,Z 185,A -30.5508,B 3.154,C 0.2566,E1 3.2962,E2 483.5867} C_DIS
LIN {X 115.9696,Y -78.5536,Z 185,A -28.9721,B 3.1542,C 0.2535,E1 3.2987,E2 482.0193} C_DIS
LIN {X 118.6551,Y -74.4362,Z 185,A -27.0933,B 3.1545,C 0.25,E1 3.3015,E2 480.1568} C_DIS
LIN {X 120.9943,Y -70.5704,Z 185,A -25.3724,B 3.1547,C 0.2467,E1 3.3039,E2 478.4516} C_DIS
LIN {X 124.4399,Y -64.3,Z 185,A -22.4478,B 3.1553,C 0.2394,E1 3.3078,E2 475.5251} C_DIS
LIN {X 126.2596,Y -60.6437,Z 185,A -20.5802,B 3.1558,C 0.233,E1 3.3101,E2 473.6294} C_DIS
LIN {X 128.0082,Y -56.8603,Z 185,A -19.2813,B 3.1558,C 0.2328,E1 3.3115,E2 472.384} C_DIS
LIN {X 129.7809,Y -52.6887,Z 185,A -17.5828,B 3.156,C 0.2295,E1 3.3133,E2 470.705} C_DIS
LIN {X 130.906,Y -49.8325,Z 185,A -15.9631,B 3.1566,C 0.2224,E1 3.315,E2 469.0353} C_DIS
LIN {X 132.2749,Y -46.0702,Z 185,A -14.6315,B 3.1566,C 0.2212,E1 3.3162,E2 467.7436} C_DIS
LIN {X 133.8293,Y -41.3394,Z 185,A -12.9004,B 3.1568,C 0.2188,E1 3.3176,E2 466.052} C_DIS
LIN {X 134.8316,Y -37.9421,Z 185,A -11.6844,B 3.1569,C 0.2173,E1 3.3186,E2 464.8659} C_DIS
LIN {X 136.5841,Y -31.0471,Z 185,A -9.0241,B 3.1573,C 0.212,E1 3.3204,E2 462.2368} C_DIS
LIN {X 137.748,Y -25.4003,Z 185,A -6.3102,B 3.1579,C 0.2017,E1 3.3219,E2 459.4742} C_DIS
LIN {X 138.2936,Y -22.242,Z 185,A -5.1755,B 3.1581,C 0.1999,E1 3.3224,E2 458.362} C_DIS
LIN {X 138.8513,Y -18.4262,Z 185,A -3.6567,B 3.1583,C 0.1961,E1 3.323,E2 456.8498} C_DIS
LIN {X 139.2525,Y -15.0974,Z 185,A -2.3439,B 3.1585,C 0.1928,E1 3.3234,E2 455.5439} C_DIS
LIN {X 139.6061,Y -11.3794,Z 185,A -0.762,B 3.1588,C 0.188,E1 3.3238,E2 453.9538} C_DIS
LIN {X 139.8882,Y -7.1066,Z 185,A 0.7732,B 3.1589,C 0.1853,E1 3.324,E2 452.446} C_DIS
LIN {X 140.0266,Y -3.4576,Z 185,A 2.2963,B 3.1592,C 0.1808,E1 3.3242,E2 450.918} C_DIS
LIN {X 140.0684,Y 0.6131,Z 185,A 3.9309,B 3.1595,C 0.1764,E1 3.3242,E2 449.2865} C_DIS
LIN {X 139.9731,Y 5.179,Z 185,A 5.6407,B 3.1597,C 0.1728,E1 3.324,E2 447.5963} C_DIS
LIN {X 139.7662,Y 9.2183,Z 185,A 7.2686,B 3.1599,C 0.1684,E1 3.3238,E2 445.9709} C_DIS
LIN {X 139.4356,Y 13.3002,Z 185,A 8.8023,B 3.1601,C 0.1652,E1 3.3234,E2 444.4547} C_DIS
LIN {X 139.0291,Y 17.0381,Z 185,A 10.3656,B 3.1603,C 0.1606,E1 3.3229,E2 442.8872} C_DIS
LIN {X 138.3612,Y 21.8054,Z 185,A 12.2398,B 3.1605,C 0.1561,E1 3.3221,E2 441.0243} C_DIS
LIN {X 137.2646,Y 27.8848,Z 185,A 14.8511,B 3.1609,C 0.1482,E1 3.3207,E2 438.4006} C_DIS
LIN {X 136.5624,Y 31.1422,Z 185,A 15.8734,B 3.1609,C 0.148,E1 3.3201,E2 437.4221} C_DIS
LIN {X 135.6185,Y 35.0297,Z 185,A 17.8516,B 3.1613,C 0.14,E1 3.3188,E2 435.3984} C_DIS
LIN {X 134.5537,Y 38.9182,Z 185,A 19.0914,B 3.1613,C 0.1397,E1 3.3178,E2 434.2113} C_DIS
LIN {X 133.4804,Y 42.4512,Z 185,A 20.4802,B 3.1614,C 0.1368,E1 3.3167,E2 432.8375} C_DIS
LIN {X 132.3734,Y 45.7864,Z 185,A 21.8272,B 3.1615,C 0.1339,E1 3.3155,E2 431.5016} C_DIS
LIN {X 131.2259,Y 48.9783,Z 185,A 23.195,B 3.1617,C 0.1304,E1 3.3142,E2 430.1358} C_DIS
LIN {X 129.9797,Y 52.1957,Z 185,A 24.5332,B 3.1618,C 0.1274,E1 3.3128,E2 428.8064} C_DIS
LIN {X 128.6292,Y 55.4403,Z 185,A 25.91,B 3.1619,C 0.1243,E1 3.3113,E2 427.4369} C_DIS
LIN {X 127.2933,Y 58.4433,Z 185,A 27.2457,B 3.1621,C 0.1209,E1 3.3098,E2 426.1018} C_DIS
LIN {X 125.7411,Y 61.7114,Z 185,A 28.5941,B 3.1621,C 0.1184,E1 3.3082,E2 424.7698} C_DIS
LIN {X 124.1348,Y 64.8819,Z 185,A 30.0247,B 3.1623,C 0.115,E1 3.3064,E2 423.3416} C_DIS
LIN {X 122.0829,Y 68.6687,Z 185,A 31.8079,B 3.1624,C 0.1104,E1 3.3039,E2 421.5551} C_DIS
LIN {X 119.7205,Y 72.7097,Z 185,A 33.6468,B 3.1626,C 0.1065,E1 3.3013,E2 419.7254} C_DIS
LIN {X 117.3089,Y 76.5398,Z 185,A 35.4433,B 3.1627,C 0.1026,E1 3.2986,E2 417.9353} C_DIS
LIN {X 114.7737,Y 80.2916,Z 185,A 37.219,B 3.1628,C 0.0989,E1 3.2958,E2 416.169} C_DIS
LIN {X 112.1227,Y 83.954,Z 185,A 38.9237,B 3.1629,C 0.0961,E1 3.293,E2 414.4824} C_DIS
LIN {X 109.7048,Y 87.0883,Z 185,A 40.8334,B 3.1631,C 0.0896,E1 3.2897,E2 412.5349} C_DIS
LIN {X 107.3206,Y 90.0105,Z 185,A 42.0628,B 3.1631,C 0.0892,E1 3.2875,E2 411.3454} C_DIS
LIN {X 104.3063,Y 93.487,Z 185,A 43.8741,B 3.1632,C 0.0858,E1 3.2842,E2 409.5428} C_DIS
LIN {X 101.1409,Y 96.9029,Z 185,A 45.6939,B 3.1632,C 0.0826,E1 3.2807,E2 407.7336} C_DIS
LIN {X 97.9752,Y 100.1024,Z 185,A 47.3738,B 3.1633,C 0.0803,E1 3.2775,E2 406.0739} C_DIS
LIN {X 94.6554,Y 103.2473,Z 185,A 49.5738,B 3.1635,C 0.0736,E1 3.2729,E2 403.8318} C_DIS
LIN {X 91.8959,Y 105.711,Z 185,A 50.6915,B 3.1635,C 0.0743,E1 3.2706,E2 402.7643} C_DIS
LIN {X 89.7576,Y 107.5329,Z 185,A 51.9341,B 3.1635,C 0.0713,E1 3.2679,E2 401.5098} C_DIS
LIN {X 86.1285,Y 110.4611,Z 185,A 53.772,B 3.1636,C 0.0685,E1 3.2639,E2 399.6805} C_DIS
LIN {X 82.5983,Y 113.1252,Z 185,A 55.4816,B 3.1636,C 0.0662,E1 3.2601,E2 397.9835} C_DIS
LIN {X 77.9296,Y 116.39,Z 185,A 57.8018,B 3.1638,C 0.0624,E1 3.2548,E2 395.6646} C_DIS
LIN {X 74.0698,Y 118.8835,Z 185,A 59.6196,B 3.1638,C 0.06,E1 3.2505,E2 393.8546} C_DIS
LIN {X 70.1531,Y 121.236,Z 185,A 61.4456,B 3.1638,C 0.0575,E1 3.2461,E2 392.0342} C_DIS
LIN {X 66.1156,Y 123.4844,Z 185,A 63.2293,B 3.1638,C 0.0557,E1 3.2418,E2 390.264} C_DIS
LIN {X 63.0684,Y 125.0668,Z 185,A 64.9407,B 3.164,C 0.0512,E1 3.2374,E2 388.514} C_DIS
LIN {X 59.5611,Y 126.7764,Z 185,A 66.2785,B 3.164,C 0.0512,E1 3.2341,E2 387.2091} C_DIS
LIN {X 55.895,Y 128.4326,Z 185,A 67.763,B 3.164,C 0.0506,E1 3.2304,E2 385.745} C_DIS
Enddeposition()
END
